	            IF ("gtyp_VGR".vertical_Axis.di_Actual_Position <= ("gtyp_VGR".di_Pos_Color_vertical + "gtyp_VGR".vertical_Axis.Config.di_Pos_Window))
	                AND ("gtyp_VGR".vertical_Axis.di_Actual_Position >= ("gtyp_VGR".di_Pos_Color_vertical - "gtyp_VGR".vertical_Axis.Config.di_Pos_Window))
	                AND "gtyp_VGR".vertical_Axis.x_Position_Reached THEN
	                "gtyp_VGR".vertical_Axis.x_Start_Positioning := FALSE;
	                "gtyp_VGR".vertical_Axis.i_PWM := 800;
	                #li_StepCase := 750;
	            END_IF;

	        750: // evaluate color workpiece
	            #ls_Color := '';

	            IF "IW_SSC_ColorSensor_A1" >= "gtyp_SSC".w_Threshold_Red_Blue THEN
	 //               IF "IW_SSC_ColorSensor" > 16000 AND "IW_SSC_ColorSensor" < 17500 THEN
	                #ls_Color := 'BLUE';
	            ELSIF "IW_SSC_ColorSensor_A1" <= "gtyp_SSC".w_Threshold_White_Red THEN
	//            ELSIF "IW_SSC_ColorSensor" > 5000 AND "IW_SSC_ColorSensor" < 11000 THEN
	                #ls_Color := 'WHITE';
	            ELSIF "IW_SSC_ColorSensor_A1" > "gtyp_SSC".w_Threshold_White_Red AND "IW_SSC_ColorSensor_A1" < "gtyp_SSC".w_Threshold_Red_Blue THEN
	//            ELSIF "IW_SSC_ColorSensor" > 11000 AND "IW_SSC_ColorSensor" < 16000 THEN
	                #ls_Color := 'RED';
	            END_IF;

	            #li_Return_LDT := RD_SYS_T(#ldt_MQTT);
	            "gtyp_VGR".History[2].ldt_ts := DT_TO_LDT(#ldt_MQTT);
	            "gtyp_VGR".History[2].i_code := 200;
	            "gtyp_VGR".Workpiece.s_type  := #ls_Color;

	            #lx_Start_TON_Wait  := TRUE;
	            #lt_TON_Wait        := T#500ms;

	            IF #lfb_TON_Wait.Q THEN
	                #lx_Start_TON_Wait := FALSE;
	                #li_StepCase := 760;
	            END_IF;

	        760: // Position vertical pre NFC
	            "gtyp_VGR".vertical_Axis.di_Target_Position := "gtyp_VGR".di_Pos_NFC_vertical - "gtyp_VGR".di_Offset_Pos_DSI_NFC_vertical;
	            "gtyp_VGR".vertical_Axis.x_Start_Positioning := TRUE;
	            "gtyp_VGR".vertical_Axis.i_PWM := 500;

	            IF ("gtyp_VGR".vertical_Axis.di_Actual_Position <= ("gtyp_VGR".di_Pos_NFC_vertical - "gtyp_VGR".di_Offset_Pos_DSI_NFC_vertical + "gtyp_VGR".vertical_Axis.Config.di_Pos_Window))
	                AND ("gtyp_VGR".vertical_Axis.di_Actual_Position >= ("gtyp_VGR".di_Pos_NFC_vertical - "gtyp_VGR".di_Offset_Pos_DSI_NFC_vertical - "gtyp_VGR".vertical_Axis.Config.di_Pos_Window))
	                AND "gtyp_VGR".vertical_Axis.x_Position_Reached THEN
	                "gtyp_VGR".vertical_Axis.x_Start_Positioning := FALSE;
	                "gtyp_VGR".vertical_Axis.i_PWM := 800;
	                #li_StepCase := 770;
	            END_IF;

	        770: // wait sequence
	            #lx_Start_TON_Wait := TRUE;
	            #lt_TON_Wait := T#500ms;

	            IF #lfb_TON_Wait.Q THEN
	                #lx_Start_TON_Wait := FALSE;
	                #li_StepCase := 780;
	            END_IF;

	        780: // Position horizontal/rotate NFC

	            "gtyp_VGR".horizontal_Axis.di_Target_Position := "gtyp_VGR".di_Pos_NFC_horizontal;
	            "gtyp_VGR".horizontal_Axis.x_Start_Positioning := TRUE;
	            "gtyp_VGR".rotate_Axis.di_Target_Position := "gtyp_VGR".di_Pos_NFC_rotate;
	            "gtyp_VGR".rotate_Axis.x_Start_Positioning := TRUE;

	            IF ("gtyp_VGR".horizontal_Axis.di_Actual_Position <= ("gtyp_VGR".di_Pos_NFC_horizontal + "gtyp_VGR".horizontal_Axis.Config.di_Pos_Window))
	                AND ("gtyp_VGR".horizontal_Axis.di_Actual_Position >= ("gtyp_VGR".di_Pos_NFC_horizontal - "gtyp_VGR".horizontal_Axis.Config.di_Pos_Window))
	                AND "gtyp_VGR".horizontal_Axis.x_Position_Reached THEN
	                "gtyp_VGR".horizontal_Axis.x_Start_Positioning := FALSE;
	            END_IF;

	            IF ("gtyp_VGR".rotate_Axis.di_Actual_Position <= ("gtyp_VGR".di_Pos_NFC_rotate + "gtyp_VGR".rotate_Axis.Config.di_Pos_Window))
	                AND ("gtyp_VGR".rotate_Axis.di_Actual_Position >= ("gtyp_VGR".di_Pos_NFC_rotate - "gtyp_VGR".rotate_Axis.Config.di_Pos_Window))
	                AND "gtyp_VGR".rotate_Axis.x_Position_Reached THEN
	                "gtyp_VGR".rotate_Axis.x_Start_Positioning := FALSE;
	            END_IF;

	            IF ("gtyp_VGR".horizontal_Axis.di_Actual_Position <= ("gtyp_VGR".di_Pos_NFC_horizontal + "gtyp_VGR".horizontal_Axis.Config.di_Pos_Window))
	                AND ("gtyp_VGR".horizontal_Axis.di_Actual_Position >= ("gtyp_VGR".di_Pos_NFC_horizontal - "gtyp_VGR".horizontal_Axis.Config.di_Pos_Window))
	                AND "gtyp_VGR".horizontal_Axis.x_Position_Reached
	                AND ("gtyp_VGR".rotate_Axis.di_Actual_Position <= ("gtyp_VGR".di_Pos_NFC_rotate + "gtyp_VGR".rotate_Axis.Config.di_Pos_Window))
	                AND ("gtyp_VGR".rotate_Axis.di_Actual_Position >= ("gtyp_VGR".di_Pos_NFC_rotate - "gtyp_VGR".rotate_Axis.Config.di_Pos_Window))
	                AND "gtyp_VGR".rotate_Axis.x_Position_Reached THEN
	                "gtyp_VGR".horizontal_Axis.x_Start_Positioning := FALSE;
	                "gtyp_VGR".vertical_Axis.x_Start_Positioning := FALSE;
	                "gtyp_VGR".rotate_Axis.x_Start_Positioning := FALSE;
	                #li_StepCase := 790;
	            END_IF;

	        790: // wait sequence
	            #lx_Start_TON_Wait := TRUE;
	            #lt_TON_Wait := T#500ms;

	            IF #lfb_TON_Wait.Q THEN
	                #lx_Start_TON_Wait := FALSE;
	                #li_StepCase := 800;
	            END_IF;

	        800: // Position vertical NFC

	            "gtyp_VGR".vertical_Axis.di_Target_Position := "gtyp_VGR".di_Pos_NFC_vertical;
	            "gtyp_VGR".vertical_Axis.x_Start_Positioning := TRUE;
	            "gtyp_VGR".vertical_Axis.i_PWM := 500;

	            IF ("gtyp_VGR".vertical_Axis.di_Actual_Position <= ("gtyp_VGR".di_Pos_NFC_vertical + "gtyp_VGR".vertical_Axis.Config.di_Pos_Window))
	                AND ("gtyp_VGR".vertical_Axis.di_Actual_Position >= ("gtyp_VGR".di_Pos_NFC_vertical - "gtyp_VGR".vertical_Axis.Config.di_Pos_Window))
	                AND "gtyp_VGR".vertical_Axis.x_Position_Reached THEN
	                "gtyp_VGR".vertical_Axis.x_Start_Positioning := FALSE;
	                "gtyp_VGR".vertical_Axis.i_PWM := 800;
	                #li_StepCase := 810;
	            END_IF;

	        810: // Start write/read NFC Color

	            "gtyp_VGR".x_NFC_Start := TRUE;

	            IF "gtyp_VGR".x_NFC_Completed THEN
	                "gtyp_VGR".x_NFC_Start := FALSE;
	                #li_StepCase := 820;
	            END_IF;

	        820: // Position vertical pre NFC

	            "gtyp_VGR".vertical_Axis.di_Target_Position := "gtyp_VGR".di_Pos_NFC_vertical - "gtyp_VGR".di_Offset_Pos_DSI_NFC_vertical;
	            "gtyp_VGR".vertical_Axis.x_Start_Positioning := TRUE;
	            "gtyp_VGR".vertical_Axis.i_PWM := 500;

	            IF ("gtyp_VGR".vertical_Axis.di_Actual_Position <= ("gtyp_VGR".di_Pos_NFC_vertical - "gtyp_VGR".di_Offset_Pos_DSI_NFC_vertical + "gtyp_VGR".vertical_Axis.Config.di_Pos_Window))
	                AND ("gtyp_VGR".vertical_Axis.di_Actual_Position >= ("gtyp_VGR".di_Pos_NFC_vertical - "gtyp_VGR".di_Offset_Pos_DSI_NFC_vertical - "gtyp_VGR".vertical_Axis.Config.di_Pos_Window))
	                AND "gtyp_VGR".vertical_Axis.x_Position_Reached THEN
	                "gtyp_VGR".vertical_Axis.x_Start_Positioning := FALSE;
	                "gtyp_VGR".vertical_Axis.i_PWM := 800;
	                #li_StepCase := 830;
	            END_IF;

	        830: // wait sequence
	            #lx_Start_TON_Wait := TRUE;
	            #lt_TON_Wait := T#500ms;

	            IF #lfb_TON_Wait.Q THEN
	                #lx_Start_TON_Wait := FALSE;
	                #li_StepCase := 840;
	            END_IF;

	        840: // Position rotate HBW and homing horizontal/vertical axis
	            "gtyp_VGR".rotate_Axis.di_Target_Position := "gtyp_VGR".di_Pos_HBW_rotate;
	            "gtyp_VGR".rotate_Axis.x_Start_Positioning := TRUE;

	            "gtyp_VGR".horizontal_Axis.x_Reference := TRUE;
	            "gtyp_VGR".vertical_Axis.x_Reference := TRUE;

	            IF ("gtyp_VGR".rotate_Axis.di_Actual_Position <= ("gtyp_VGR".di_Pos_HBW_rotate + "gtyp_VGR".rotate_Axis.Config.di_Pos_Window))
	                AND ("gtyp_VGR".rotate_Axis.di_Actual_Position >= ("gtyp_VGR".di_Pos_HBW_rotate - "gtyp_VGR".rotate_Axis.Config.di_Pos_Window))
	                AND "gtyp_VGR".rotate_Axis.x_Position_Reached THEN
	                "gtyp_VGR".rotate_Axis.x_Start_Positioning := FALSE;
	            END_IF;

	            IF NOT "gtyp_VGR".horizontal_Axis.x_Referenced AND NOT "gtyp_VGR".vertical_Axis.x_Referenced THEN
	                #li_StepCase := 850;
	            END_IF;

	        850: // Position rotate HBW reached and homed horizontal/vertical axis

	            IF ("gtyp_VGR".rotate_Axis.di_Actual_Position <= ("gtyp_VGR".di_Pos_HBW_rotate + "gtyp_VGR".rotate_Axis.Config.di_Pos_Window))
	                AND ("gtyp_VGR".rotate_Axis.di_Actual_Position >= ("gtyp_VGR".di_Pos_HBW_rotate - "gtyp_VGR".rotate_Axis.Config.di_Pos_Window))
	                AND "gtyp_VGR".rotate_Axis.x_Position_Reached THEN
	                "gtyp_VGR".rotate_Axis.x_Start_Positioning := FALSE;
	            END_IF;

	            IF "gtyp_VGR".horizontal_Axis.x_Referenced THEN
	                "gtyp_VGR".horizontal_Axis.x_Reference := FALSE;
	            END_IF;
	            IF "gtyp_VGR".vertical_Axis.x_Referenced THEN
	                "gtyp_VGR".vertical_Axis.x_Reference := FALSE;
	            END_IF;
	            IF "gtyp_VGR".horizontal_Axis.x_Referenced
	                AND "gtyp_VGR".vertical_Axis.x_Referenced
	                AND ("gtyp_VGR".rotate_Axis.di_Actual_Position <= ("gtyp_VGR".di_Pos_HBW_rotate + "gtyp_VGR".rotate_Axis.Config.di_Pos_Window))
	                AND ("gtyp_VGR".rotate_Axis.di_Actual_Position >= ("gtyp_VGR".di_Pos_HBW_rotate - "gtyp_VGR".rotate_Axis.Config.di_Pos_Window))
	                AND "gtyp_VGR".rotate_Axis.x_Position_Reached THEN
	                "gtyp_VGR".horizontal_Axis.x_Reference := FALSE;
	                "gtyp_VGR".vertical_Axis.x_Reference := FALSE;
	                "gtyp_VGR".rotate_Axis.x_Start_Positioning := FALSE;
	                #li_StepCase := 860;
	            END_IF;

	        860: // wait sequence
	            #lx_Start_TON_Wait := TRUE;
	            #lt_TON_Wait := T#500ms;

	            IF #lfb_TON_Wait.Q THEN
	                #lx_Start_TON_Wait := FALSE;
	                #li_StepCase := 870;
	            END_IF;

	        870: // Position horizontal HBW

	            "gtyp_VGR".horizontal_Axis.di_Target_Position := "gtyp_VGR".di_Pos_HBW_horizontal;
	            "gtyp_VGR".horizontal_Axis.x_Start_Positioning := TRUE;

	            IF ("gtyp_VGR".horizontal_Axis.di_Actual_Position <= ("gtyp_VGR".di_Pos_HBW_horizontal + "gtyp_VGR".horizontal_Axis.Config.di_Pos_Window))
	                AND ("gtyp_VGR".horizontal_Axis.di_Actual_Position >= ("gtyp_VGR".di_Pos_HBW_horizontal - "gtyp_VGR".horizontal_Axis.Config.di_Pos_Window))
	                AND "gtyp_VGR".horizontal_Axis.x_Position_Reached THEN
	                "gtyp_VGR".horizontal_Axis.x_Start_Positioning := FALSE;
	                #li_StepCase := 880;
	            END_IF;

	        880: // container available start drop down
	            IF "gtyp_HBW".x_HBW_Container_Available THEN
	                #li_StepCase := 890;
	            END_IF;

	        890: // Position vertical discard HBW
	            "gtyp_VGR".vertical_Axis.di_Target_Position := "gtyp_VGR".di_Pos_HBW_Discard_vertical;
	            "gtyp_VGR".vertical_Axis.x_Start_Positioning := TRUE;
	            "gtyp_VGR".vertical_Axis.i_PWM := 500;

	            IF ("gtyp_VGR".vertical_Axis.di_Actual_Position <= ("gtyp_VGR".di_Pos_HBW_Discard_vertical + "gtyp_VGR".vertical_Axis.Config.di_Pos_Window))
	                AND ("gtyp_VGR".vertical_Axis.di_Actual_Position >= ("gtyp_VGR".di_Pos_HBW_Discard_vertical - "gtyp_VGR".vertical_Axis.Config.di_Pos_Window))
	                AND "gtyp_VGR".vertical_Axis.x_Position_Reached THEN
	                "gtyp_VGR".vertical_Axis.x_Start_Positioning := FALSE;
	                "gtyp_VGR".vertical_Axis.i_PWM := 800;
	                #li_StepCase := 900;
	            END_IF;

	        900: // turn off vacuum
	            "QX_VGR_ValveVacuum_Q8" := FALSE;
	            #li_StepCase := 910;

	        910: // turn off compressor
	            "QX_VGR_Compressor_Q7" := FALSE;
	            "gtyp_VGR".x_HBW_Discards := TRUE;

	            #lx_Start_TON_Wait := TRUE;
	            #lt_TON_Wait := T#500ms;

	            IF #lfb_TON_Wait.Q AND "gtyp_HBW".x_HBW_Discards_Accepted THEN
	                #lx_State_activ := FALSE;
	                #ls_Target := '';
	                "gtyp_VGR".x_HBW_Discards   := FALSE;
	                "gtyp_VGR".x_HBW_Storage  := FALSE;
	                #lx_Start_TON_Wait                   := FALSE;
	                #li_StepCase                := 920;
	            END_IF;

	        920: // homing vertical axis
	            "gtyp_VGR".vertical_Axis.x_Reference := TRUE;

	            IF NOT "gtyp_VGR".vertical_Axis.x_Referenced THEN
	                #li_StepCase := 930;
	            END_IF;

	        930: // homed vertical axis
	            IF "gtyp_VGR".vertical_Axis.x_Referenced THEN
	                "gtyp_VGR".vertical_Axis.x_Reference := FALSE;
	                #li_StepCase := 940;
	            END_IF;

	        940: // homing horizontal axis
	            "gtyp_VGR".horizontal_Axis.x_Reference := TRUE;

	            IF NOT "gtyp_VGR".horizontal_Axis.x_Referenced THEN
	                #li_StepCase := 950;
	            END_IF;

	        950: // homed horizontal axis
	            IF "gtyp_VGR".horizontal_Axis.x_Referenced THEN
	                "gtyp_VGR".horizontal_Axis.x_Reference := FALSE;
	                #li_StepCase := 960;
	            END_IF;

	        960: // wait sequence
	            #lx_Start_TON_Wait := TRUE;
	            #lt_TON_Wait := T#500ms;

	            IF #lfb_TON_Wait.Q AND "gtyp_HBW".x_HBW_Discards_Accepted THEN
	                "gtyp_VGR".x_HBW_Discards  := FALSE;
	                #lx_Start_TON_Wait               := FALSE;
	                "gtyp_VGR".Workpiece.s_id       := '';
	                "gtyp_VGR".Workpiece.s_state    := '';
	                "gtyp_VGR".Workpiece.s_type     := '';
	                FOR #li_Counter := 1 TO 8 DO
	                    // Statement section FOR
	                    "gtyp_VGR".History[#li_Counter].i_code := 0;
	                    "gtyp_VGR".History[#li_Counter].ldt_ts := DT#1990-01-01-00:00:00;
	                END_FOR;
	                #li_StepCase := 0;
	            END_IF;

	        1200:// homing vertical axis
	            "gtyp_VGR".Workpiece.s_id := '0';
	            "gtyp_VGR".Workpiece.s_state := '';
	            "gtyp_VGR".Workpiece.s_type := '';
	            FOR #li_Counter := 1 TO 8 DO
	                "gtyp_VGR".History[#li_Counter].i_code := 0;
	                "gtyp_VGR".History[#li_Counter].ldt_ts := DT#1990-01-01-00:00:00;
	            END_FOR;

	            IF "gtyp_HBW".x_HBW_Container_Available THEN
	                "gtyp_VGR".x_HBW_Discards := TRUE;
	            END_IF;

	            IF "gtyp_HBW".x_HBW_Discards_Accepted OR "gtyp_HBW".x_HBW_PickedUp_Accepted THEN
	                "gtyp_VGR".x_HBW_Discards := FALSE;
	                "gtyp_VGR".x_HBW_PickedUp := FALSE;
	                "gtyp_HBW".x_HBW_Discards_Accepted := FALSE;
	                "gtyp_HBW".x_HBW_PickedUp_Accepted := FALSE;
	            END_IF;

	            #li_Lights := 2;
	            "gtyp_VGR".vertical_Axis.x_Reference := TRUE;

	            IF NOT "gtyp_VGR".vertical_Axis.x_Referenced THEN
	                #li_StepCase := 1210;
	            END_IF;

	        1210: // homed vertical axis
	            IF "gtyp_VGR".vertical_Axis.x_Referenced THEN
	                "gtyp_VGR".vertical_Axis.x_Reference := FALSE;
	                #li_StepCase := 1220;
	            END_IF;

	        1220: // homing horizontal axis
	            "gtyp_VGR".horizontal_Axis.x_Reference := TRUE;

	            IF NOT "gtyp_VGR".horizontal_Axis.x_Referenced THEN
	                #li_StepCase := 1230;
	            END_IF;

	        1230: // homed horizontal axis
	            IF "gtyp_VGR".horizontal_Axis.x_Referenced THEN
	                "gtyp_VGR".horizontal_Axis.x_Reference := FALSE;
	                #li_StepCase := 1240;
	            END_IF;

	        1240: // homing rotate axis
	            "gtyp_VGR".rotate_Axis.x_Reference := TRUE;

	            IF NOT "gtyp_VGR".rotate_Axis.x_Referenced THEN
	                #li_StepCase := 1250;
	            END_IF;

	        1250: // homed horizontal axis
	            IF "gtyp_VGR".rotate_Axis.x_Referenced THEN
	                "gtyp_VGR".rotate_Axis.x_Reference := FALSE;
	                #li_StepCase := 1260;
	            END_IF;

	        1260: // Position vertical/horizontal/rotate NiO
	            "gtyp_VGR".horizontal_Axis.di_Target_Position := "gtyp_VGR".di_Pos_NiO_horizontal;
	            "gtyp_VGR".horizontal_Axis.x_Start_Positioning := TRUE;
	            "gtyp_VGR".vertical_Axis.di_Target_Position := "gtyp_VGR".di_Pos_NiO_vertical;
	            "gtyp_VGR".vertical_Axis.x_Start_Positioning := TRUE;
	            "gtyp_VGR".vertical_Axis.i_PWM := 500;
	            "gtyp_VGR".rotate_Axis.di_Target_Position := "gtyp_VGR".di_Pos_NiO_rotate;
	            "gtyp_VGR".rotate_Axis.x_Start_Positioning := TRUE;

	            IF ("gtyp_VGR".horizontal_Axis.di_Actual_Position <= ("gtyp_VGR".di_Pos_NiO_horizontal + "gtyp_VGR".horizontal_Axis.Config.di_Pos_Window))
	                AND ("gtyp_VGR".horizontal_Axis.di_Actual_Position >= ("gtyp_VGR".di_Pos_NiO_horizontal - "gtyp_VGR".horizontal_Axis.Config.di_Pos_Window))
	                AND "gtyp_VGR".horizontal_Axis.x_Position_Reached THEN
	                "gtyp_VGR".horizontal_Axis.x_Start_Positioning := FALSE;
	            END_IF;

	            IF ("gtyp_VGR".vertical_Axis.di_Actual_Position <= ("gtyp_VGR".di_Pos_NiO_vertical + "gtyp_VGR".vertical_Axis.Config.di_Pos_Window))
	                AND ("gtyp_VGR".vertical_Axis.di_Actual_Position >= ("gtyp_VGR".di_Pos_NiO_vertical - "gtyp_VGR".vertical_Axis.Config.di_Pos_Window))
	                AND "gtyp_VGR".vertical_Axis.x_Position_Reached THEN
	                "gtyp_VGR".vertical_Axis.x_Start_Positioning := FALSE;
	            END_IF;

	            IF ("gtyp_VGR".rotate_Axis.di_Actual_Position <= ("gtyp_VGR".di_Pos_NiO_rotate + "gtyp_VGR".rotate_Axis.Config.di_Pos_Window))
	                AND ("gtyp_VGR".rotate_Axis.di_Actual_Position >= ("gtyp_VGR".di_Pos_NiO_rotate - "gtyp_VGR".rotate_Axis.Config.di_Pos_Window))
	                AND "gtyp_VGR".rotate_Axis.x_Position_Reached THEN
	                "gtyp_VGR".rotate_Axis.x_Start_Positioning := FALSE;
	            END_IF;

	            IF ("gtyp_VGR".horizontal_Axis.di_Actual_Position <= ("gtyp_VGR".di_Pos_NiO_horizontal + "gtyp_VGR".horizontal_Axis.Config.di_Pos_Window))
	                AND ("gtyp_VGR".horizontal_Axis.di_Actual_Position >= ("gtyp_VGR".di_Pos_NiO_horizontal - "gtyp_VGR".horizontal_Axis.Config.di_Pos_Window))
	                AND "gtyp_VGR".horizontal_Axis.x_Position_Reached
	                AND ("gtyp_VGR".vertical_Axis.di_Actual_Position <= ("gtyp_VGR".di_Pos_NiO_vertical + "gtyp_VGR".vertical_Axis.Config.di_Pos_Window))
	                AND ("gtyp_VGR".vertical_Axis.di_Actual_Position >= ("gtyp_VGR".di_Pos_NiO_vertical - "gtyp_VGR".vertical_Axis.Config.di_Pos_Window))
	                AND "gtyp_VGR".vertical_Axis.x_Position_Reached
	                AND ("gtyp_VGR".rotate_Axis.di_Actual_Position <= ("gtyp_VGR".di_Pos_NiO_rotate + "gtyp_VGR".rotate_Axis.Config.di_Pos_Window))
	                AND ("gtyp_VGR".rotate_Axis.di_Actual_Position >= ("gtyp_VGR".di_Pos_NiO_rotate - "gtyp_VGR".rotate_Axis.Config.di_Pos_Window))
	                AND "gtyp_VGR".rotate_Axis.x_Position_Reached THEN
	                "gtyp_VGR".horizontal_Axis.x_Start_Positioning := FALSE;
	                "gtyp_VGR".vertical_Axis.x_Start_Positioning := FALSE;
	                "gtyp_VGR".rotate_Axis.x_Start_Positioning := FALSE;
	                "gtyp_VGR".vertical_Axis.i_PWM := 800;
	                #li_StepCase := 1270;
	            END_IF;

	        1270: // turn off vacuum
	            "QX_VGR_ValveVacuum_Q8" := FALSE;
	            #li_StepCase := 1280;

	        1280: // turn off compressor

	            #lx_Start_TON_Wait := TRUE;
	            #lt_TON_Wait := T#1000ms;

	            IF #lfb_TON_Wait.Q THEN
	                "QX_VGR_Compressor_Q7"  := FALSE;
	                #lx_Start_TON_Wait               := FALSE;
	                "gtyp_VGR".x_Workpiece_NiO := FALSE;
	                "gtyp_VGR".x_HBW_Discards := FALSE;
	                #li_Lights := 1;
	                #li_StepCase            := 0;
	            END_IF;
	    // Statement section ELSE
	    ELSE
	            ;
	    END_CASE;

	ELSE
	    "gtyp_VGR".Workpiece.s_id := '';
	    "gtyp_VGR".Workpiece.s_state := '';
	    "gtyp_VGR".Workpiece.s_type := '';
	    // Order State
	    "gtyp_VGR".x_State_Process := FALSE;
	    "gtyp_Interface_Dashboard".Subscribe.State_Order.ldt_ts := DT_TO_LDT(#ldt_MQTT);
	    "gtyp_Interface_Dashboard".Subscribe.State_Order.s_state := 'WAITING_FOR_ORDER';
	    "gtyp_Interface_Dashboard".Subscribe.State_Order.s_type := '';
	    FOR #li_Counter := 1 TO 8 DO
	        "gtyp_VGR".History[#li_Counter].i_code := 0;
	        "gtyp_VGR".History[#li_Counter].ldt_ts := DT#1990-01-01-00:00:00;
	    END_FOR;

	    "gtyp_VGR".x_Start_Park_Position    := FALSE;
	    "gtyp_VGR".x_Park_Position_Reached  := FALSE;
	    "gtyp_VGR".x_NFC_Start_First        := FALSE;
	    "gtyp_VGR".x_NFC_Start              := FALSE;
	    "gtyp_VGR".x_NFC_Completed          := FALSE;
	    "gtyp_VGR".x_HBW_Storage            := FALSE;
	    "gtyp_VGR".x_HBW_Outsource          := FALSE;
	    "gtyp_VGR".s_HBW_Outsource_Typ      := '';
	    "gtyp_VGR".x_HBW_Discards           := FALSE;
	    "gtyp_VGR".x_HBW_PickedUp           := FALSE;
	    "gtyp_VGR".x_MPO_Req_Discard        := FALSE;
	    "gtyp_VGR".x_MPO_Discards           := FALSE;
	    "gtyp_VGR".x_Ready_For_Outsource    := FALSE;
	    "gtyp_VGR".x_State_Process          := FALSE;
	    "gtyp_VGR".x_Workpiece_NiO          := FALSE;

	    "gtyp_VGR".vertical_Axis.i_PWM      := 800;

	    #li_Lights := 1;
	    #lx_Init := TRUE;
	END_IF;
END_FUNCTION_BLOCK

FUNCTION_BLOCK "PRG_Order"
TITLE = Program Order
{ S7_Optimized_Access := 'TRUE' }
AUTHOR : 'A.Schaefer'
VERSION : 0.0
   VAR
      lx_Init { ExternalAccessible := 'False'; ExternalVisible := 'False'; ExternalWritable := 'False'} : Bool;
      li_StepCase { ExternalAccessible := 'False'; ExternalVisible := 'False'; ExternalWritable := 'False'} : Int;
      lldt_ts_old { ExternalAccessible := 'False'; ExternalVisible := 'False'; ExternalWritable := 'False'} : LDT;
      ldt_MQTT { ExternalAccessible := 'False'; ExternalVisible := 'False'; ExternalWritable := 'False'} : Date_And_Time;
      li_Return_LDT { ExternalAccessible := 'False'; ExternalVisible := 'False'; ExternalWritable := 'False'} : Int;
      lfb_TON_Wait {InstructionName := 'TON_TIME'; LibVersion := '1.0'; ExternalAccessible := 'False'; ExternalVisible := 'False'; ExternalWritable := 'False'; S7_SetPoint := 'False'} : TON_TIME;
      lx_Start_TON_Wait { ExternalAccessible := 'False'; ExternalVisible := 'False'; ExternalWritable := 'False'} : Bool;
   END_VAR


BEGIN
	IF #lx_Init THEN
	    #lfb_TON_Wait(IN:= #lx_Start_TON_Wait,PT:= T#20s);

	    // step chain order
	    CASE #li_StepCase OF

	        0:  // init
	            #lx_Start_TON_Wait := FALSE;
	            #li_StepCase := 10;

	        10: // check whether order button has been pressed (time stamp changes)
	            IF ("gtyp_Interface_Dashboard".Publish.OrderWorkpieceButton.ldt_ts > #lldt_ts_old) THEN
	                #li_Return_LDT := RD_SYS_T(#ldt_MQTT);
	                "gtyp_Interface_Dashboard".Subscribe.State_Order.ldt_ts := DT_TO_LDT(#ldt_MQTT);
	                "gtyp_Interface_Dashboard".Subscribe.State_Order.s_state := 'ORDERED';
	                "gtyp_VGR".s_HBW_Outsource_Typ := "gtyp_Interface_Dashboard".Publish.OrderWorkpieceButton.s_type;
	                "gtyp_Interface_Dashboard".Subscribe.State_Order.s_type := "gtyp_VGR".s_HBW_Outsource_Typ;
	                IF "gtyp_VGR".x_Ready_For_Outsource THEN
	                    #lldt_ts_old := "gtyp_Interface_Dashboard".Publish.OrderWorkpieceButton.ldt_ts;
	                    "gtyp_VGR".x_HBW_Outsource := TRUE;
	                    #li_StepCase := 20;
	                END_IF;
	            END_IF;

	        20: // delete
	            IF "gtyp_VGR".x_HBW_PickedUp OR NOT "gtyp_VGR".x_HBW_Outsource THEN
	                "gtyp_VGR".x_HBW_Outsource := FALSE;
	                "gtyp_VGR".s_HBW_Outsource_Typ := '';
	                #li_StepCase := 0;
	            END_IF;

	    // Statement section ELSE
	    ELSE
	                ;
	    END_CASE;

	ELSE
	    #lx_Init    := TRUE;
	    #lldt_ts_old:= LDT#1970-01-01-00:00:00;
	END_IF;
END_FUNCTION_BLOCK

FUNCTION_BLOCK "PRG_MPO_Set_Park_Position"
TITLE = Program Set Positioning HBW
{ S7_Optimized_Access := 'TRUE' }
AUTHOR : 'A.Schaefer'
VERSION : 0.0
   VAR
      lx_Init { ExternalAccessible := 'False'; ExternalVisible := 'False'; ExternalWritable := 'False'} : Bool;
      lx_Start_TON_Wait { ExternalAccessible := 'False'; ExternalVisible := 'False'; ExternalWritable := 'False'} : Bool;
      lt_TON_Wait { ExternalAccessible := 'False'; ExternalVisible := 'False'; ExternalWritable := 'False'} : Time;
      li_StepCase { ExternalAccessible := 'False'; ExternalVisible := 'False'; ExternalWritable := 'False'} : Int;
      lfb_TON_Wait {InstructionName := 'TON_TIME'; LibVersion := '1.0'; ExternalAccessible := 'False'; ExternalVisible := 'False'; ExternalWritable := 'False'; S7_SetPoint := 'False'} : TON_TIME;
      lfb_R_Trig_Start_Park_Pos {InstructionName := 'R_TRIG'; LibVersion := '1.0'; ExternalAccessible := 'False'; ExternalVisible := 'False'; ExternalWritable := 'False'; S7_SetPoint := 'False'} : R_TRIG;
   END_VAR


BEGIN
	IF #lx_Init THEN

	    // FB TON Wait
	    #lfb_TON_Wait(IN := #lx_Start_TON_Wait,
	                  PT := #lt_TON_Wait);

	    #lfb_R_Trig_Start_Park_Pos(CLK := "gtyp_Setup".x_Park_Position
	                               OR "IX_Set_Park_Position");

	    // Set Start Park Position
	    IF #lfb_R_Trig_Start_Park_Pos.Q THEN
	        "gtyp_MPO".x_Start_Park_Position := TRUE;
	        #li_StepCase := 0;
	    END_IF;

	    // not Start Park Pos Step 0
	    IF NOT "gtyp_MPO".x_Start_Park_Position THEN
	        #li_StepCase := 0;
	    END_IF;

	    // step chain HBW
	    CASE #li_StepCase OF

	        0:  // init
	            #lx_Start_TON_Wait := FALSE;
	            #li_StepCase := 10;

	        10:  // Set Positioning activ?
	            IF "gtyp_MPO".x_Start_Park_Position AND NOT "gtyp_MPO".x_Park_Position_Reached THEN
	                #li_StepCase := 20;
	            END_IF;

	        20: // Towards
	            "QX_MPO_M5_VacuumTowardsTurnTable_Q8" := FALSE;
	            "QX_MPO_M5_VacuumTowardsOven_Q7"    := TRUE;
	            #lx_Start_TON_Wait                  := TRUE;
	            #lt_TON_Wait                        := T#4000ms;

	            IF #lfb_TON_Wait.Q THEN
	                "QX_MPO_M5_VacuumTowardsTurnTable_Q8" := FALSE;
	                "QX_MPO_M5_VacuumTowardsOven_Q7"    := FALSE;
	                #lx_Start_TON_Wait                  := FALSE;
	                #li_StepCase                        := 30;
	            END_IF;

	        30: // homing vertical axis
	            "QX_MPO_M1_TurnTableClockwise_Q1"        := TRUE;
	            "QX_MPO_M1_TurnTableCounterclockwise_Q2" := FALSE;
	            #lx_Start_TON_Wait := TRUE;
	            #lt_TON_Wait := T#1000ms;

	            IF #lfb_TON_Wait.Q THEN
	                "QX_MPO_M1_TurnTableClockwise_Q1" := FALSE;
	                "QX_MPO_M1_TurnTableCounterclockwise_Q2" := FALSE;
	                #lx_Start_TON_Wait := FALSE;
	                #li_StepCase := 40;
	            END_IF;

	        40: // Deciding which doing
	            "gtyp_MPO".x_Park_Position_Reached := TRUE;


	            // Statement section ELSE
	        ELSE
	            ;
	    END_CASE;

	ELSE
	    #lx_Init := TRUE;
	END_IF;
END_FUNCTION_BLOCK

FUNCTION_BLOCK "PRG_HBW_Ablauf"
TITLE = Program Ablauf HBW
{ S7_Optimized_Access := 'TRUE' }
AUTHOR : 'A.Schaefer'
VERSION : 0.0
   VAR
      lx_Init { ExternalAccessible := 'False'; ExternalVisible := 'False'; ExternalWritable := 'False'} : Bool;
      lx_Start_TON_Wait { ExternalAccessible := 'False'; ExternalVisible := 'False'; ExternalWritable := 'False'} : Bool;
      lx_Time_Error { ExternalAccessible := 'False'; ExternalVisible := 'False'; ExternalWritable := 'False'} : Bool;
      lt_TON_Wait { ExternalAccessible := 'False'; ExternalVisible := 'False'; ExternalWritable := 'False'} : Time;
      lx_Start_TON_State { ExternalAccessible := 'False'; ExternalVisible := 'False'; ExternalWritable := 'False'} : Bool;
      lx_Storage { ExternalAccessible := 'False'; ExternalVisible := 'False'; ExternalWritable := 'False'} : Bool;
      ldt_MQTT { ExternalAccessible := 'False'; ExternalVisible := 'False'; ExternalWritable := 'False'} : Date_And_Time;
      li_Return_LDT { ExternalAccessible := 'False'; ExternalVisible := 'False'; ExternalWritable := 'False'} : Int;
      lldt_Outsource { ExternalAccessible := 'False'; ExternalVisible := 'False'; ExternalWritable := 'False'} : LDT;
      li_Lights { ExternalAccessible := 'False'; ExternalVisible := 'False'; ExternalWritable := 'False'} : Int;
      li_Lights_old { ExternalAccessible := 'False'; ExternalVisible := 'False'; ExternalWritable := 'False'} : Int;
      li_Counter_Hor { ExternalAccessible := 'False'; ExternalVisible := 'False'; ExternalWritable := 'False'} : Int;
      li_Counter_Ver { ExternalAccessible := 'False'; ExternalVisible := 'False'; ExternalWritable := 'False'} : Int;
      li_Counter_Act_Hor { ExternalAccessible := 'False'; ExternalVisible := 'False'; ExternalWritable := 'False'} : Int;
      li_Counter_Act_Ver { ExternalAccessible := 'False'; ExternalVisible := 'False'; ExternalWritable := 'False'} : Int;
      li_Counter { ExternalAccessible := 'False'; ExternalVisible := 'False'; ExternalWritable := 'False'} : Int;
      li_StepCase { ExternalAccessible := 'False'; ExternalVisible := 'False'; ExternalWritable := 'False'} : Int;
      ldi_PosRack_Horizontal { ExternalAccessible := 'False'; ExternalVisible := 'False'; ExternalWritable := 'False'} : DInt;
      ldi_PosRack_Vertical { ExternalAccessible := 'False'; ExternalVisible := 'False'; ExternalWritable := 'False'} : DInt;
      ls_Color { ExternalAccessible := 'False'; ExternalVisible := 'False'; ExternalWritable := 'False'} : String;
      lfb_TON_State {InstructionName := 'TON_TIME'; LibVersion := '1.0'; ExternalAccessible := 'False'; ExternalVisible := 'False'; ExternalWritable := 'False'; S7_SetPoint := 'False'} : TON_TIME;
      lfb_TON_ConveyerBelt_Out {InstructionName := 'TON_TIME'; LibVersion := '1.0'; ExternalAccessible := 'False'; ExternalVisible := 'False'; ExternalWritable := 'False'; S7_SetPoint := 'False'} : TON_TIME;
      lfb_TON_Wait {InstructionName := 'TON_TIME'; LibVersion := '1.0'; ExternalAccessible := 'False'; ExternalVisible := 'False'; ExternalWritable := 'False'; S7_SetPoint := 'False'} : TON_TIME;
      lfb_TON_Error {InstructionName := 'TON_TIME'; LibVersion := '1.0'; ExternalAccessible := 'False'; ExternalVisible := 'False'; ExternalWritable := 'False'; S7_SetPoint := 'False'} : TON_TIME;
   END_VAR


BEGIN
	IF #lx_Init THEN

	    // Restart after set Positioning
	    IF "gtyp_Setup".x_Set_Pos_Activ OR "gtyp_HBW".x_Start_Park_Position THEN
	        #li_StepCase := 0;
	    END_IF;

	    // wait time state
	    #lfb_TON_State(IN := NOT #lx_Start_TON_State,
	                    PT := T#2s);

	    // runtime monitoring error
	    #lfb_TON_Error(IN := #lx_Time_Error,
	                   PT := T#30s);

	    // state of the Stock HBW cyclically transmitted to the cloud
	     IF (#lfb_TON_State.Q OR (#li_Lights <> #li_Lights_old)) AND NOT #lx_Start_TON_State THEN
	        #li_Lights_old := #li_Lights;
	        #lx_Start_TON_State := TRUE;
	        #li_Return_LDT := RD_SYS_T(#ldt_MQTT);
	        "gtyp_Interface_Dashboard".Subscribe.Stock_HBW.StockItem := "gtyp_HBW".Rack_Workpiece;
	        "gtyp_Interface_Dashboard".Subscribe.Stock_HBW.ldt_ts := DT_TO_LDT(#ldt_MQTT);

	        "gtyp_Interface_Dashboard".Subscribe.State_HBW.ldt_ts := DT_TO_LDT(#ldt_MQTT);
	        "gtyp_Interface_Dashboard".Subscribe.State_HBW.i_code := #li_Lights;
	        "gtyp_Interface_Dashboard".Subscribe.State_HBW.s_description := '';
	        "gtyp_Interface_Dashboard".Subscribe.State_HBW.s_station := 'hbw';
	        "gtyp_Interface_Dashboard".Subscribe.State_HBW.s_target := '';
	    END_IF;

	    // restart wait time state
	    IF NOT #lfb_TON_State.Q AND #lx_Start_TON_State THEN
	        #lx_Start_TON_State := FALSE;
	    END_IF;

	    // FB TON Wait
	    #lfb_TON_Wait(IN := #lx_Start_TON_Wait,
	                    PT := #lt_TON_Wait);

	    //Run-on time Conveyer Belt
	    #lfb_TON_ConveyerBelt_Out(IN := NOT "IX_HBW_LightBarrierOutside_I3",
	                              PT := T#300ms);

	    // Reload the calibration values - Rack Array
	    // A
	    "gtyp_HBW".Rack_Pos[1, 1].di_PosRack_Horizontal := "gtyp_HBW".di_PosRack_A1_Horizontal;
	    "gtyp_HBW".Rack_Pos[2, 1].di_PosRack_Horizontal := "gtyp_HBW".di_PosRack_A1_Horizontal;
	    "gtyp_HBW".Rack_Pos[3, 1].di_PosRack_Horizontal := "gtyp_HBW".di_PosRack_A1_Horizontal;
	    // B
	    "gtyp_HBW".Rack_Pos[1, 2].di_PosRack_Horizontal := "gtyp_HBW".di_PosRack_B2_Horizontal;
	    "gtyp_HBW".Rack_Pos[2, 2].di_PosRack_Horizontal := "gtyp_HBW".di_PosRack_B2_Horizontal;
	    "gtyp_HBW".Rack_Pos[3, 2].di_PosRack_Horizontal := "gtyp_HBW".di_PosRack_B2_Horizontal;
	    // C
	    "gtyp_HBW".Rack_Pos[1, 3].di_PosRack_Horizontal := "gtyp_HBW".di_PosRack_C3_Horizontal;
	    "gtyp_HBW".Rack_Pos[2, 3].di_PosRack_Horizontal := "gtyp_HBW".di_PosRack_C3_Horizontal;
	    "gtyp_HBW".Rack_Pos[3, 3].di_PosRack_Horizontal := "gtyp_HBW".di_PosRack_C3_Horizontal;
	    // 1
	    "gtyp_HBW".Rack_Pos[1, 1].di_PosRack_Vertical := "gtyp_HBW".di_PosRack_A1_Vertical;
	    "gtyp_HBW".Rack_Pos[1, 2].di_PosRack_Vertical := "gtyp_HBW".di_PosRack_A1_Vertical;
	    "gtyp_HBW".Rack_Pos[1, 3].di_PosRack_Vertical := "gtyp_HBW".di_PosRack_A1_Vertical;
	    // 2
	    "gtyp_HBW".Rack_Pos[2, 1].di_PosRack_Vertical := "gtyp_HBW".di_PosRack_B2_Vertical;
	    "gtyp_HBW".Rack_Pos[2, 2].di_PosRack_Vertical := "gtyp_HBW".di_PosRack_B2_Vertical;
	    "gtyp_HBW".Rack_Pos[2, 3].di_PosRack_Vertical := "gtyp_HBW".di_PosRack_B2_Vertical;
	    // 3
	    "gtyp_HBW".Rack_Pos[3, 1].di_PosRack_Vertical := "gtyp_HBW".di_PosRack_C3_Vertical;
	    "gtyp_HBW".Rack_Pos[3, 2].di_PosRack_Vertical := "gtyp_HBW".di_PosRack_C3_Vertical;
	    "gtyp_HBW".Rack_Pos[3, 3].di_PosRack_Vertical := "gtyp_HBW".di_PosRack_C3_Vertical;

	    // step chain HBW
	    CASE #li_StepCase OF

	        0:  // init
	            #lx_Start_TON_Wait := FALSE;
	            #lx_Time_Error := FALSE;

	            "gtyp_HBW".Horizontal_Axis.x_Start_Positioning := FALSE;
	            "gtyp_HBW".Vertical_Axis.x_Start_Positioning := FALSE;
	            "gtyp_HBW".Horizontal_Axis.x_Reference := FALSE;
	            "gtyp_HBW".Vertical_Axis.x_Reference := FALSE;

	            IF NOT "gtyp_HBW".x_Error AND NOT "gtyp_Setup".x_Set_Pos_Activ AND NOT "gtyp_HBW".x_Start_Park_Position THEN
	                #li_StepCase := 10;
	            END_IF;

	        10:  // Position Cantilever Back
	            #li_Lights := 2;
	            IF "IX_HBW_SwitchCantileverFront_I5" OR NOT "IX_HBW_SwitchCantileverBack_I6" THEN
	                "QX_HBW_M4_CantileverBackward_Q8" := TRUE;
	                "QX_HBW_M4_CantileverForward_Q7" := FALSE;
	            ELSIF NOT "IX_HBW_SwitchCantileverFront_I5" AND "IX_HBW_SwitchCantileverBack_I6" THEN
	                "QX_HBW_M4_CantileverBackward_Q8" := FALSE;
	                "QX_HBW_M4_CantileverForward_Q7" := FALSE;
	                #li_StepCase := 20;
	            END_IF;

	        20: //homing vertical/horizontal axis

	            "gtyp_HBW".Horizontal_Axis.x_Reference := TRUE;
	            "gtyp_HBW".Vertical_Axis.x_Reference := TRUE;

	            IF NOT "gtyp_HBW".Horizontal_Axis.x_Referenced AND NOT "gtyp_HBW".Vertical_Axis.x_Referenced THEN
	                #li_StepCase := 30;
	            END_IF;

	        30: // homed vertical/horizontal axis
	            IF "gtyp_HBW".Horizontal_Axis.x_Referenced THEN
	                "gtyp_HBW".Horizontal_Axis.x_Reference := FALSE;
	            END_IF;
	            IF "gtyp_HBW".Vertical_Axis.x_Referenced THEN
	                "gtyp_HBW".Vertical_Axis.x_Reference := FALSE;
	            END_IF;

	            IF "gtyp_HBW".Horizontal_Axis.x_Referenced AND "gtyp_HBW".Vertical_Axis.x_Referenced THEN
	                "gtyp_HBW".Horizontal_Axis.x_Reference := FALSE;
	                "gtyp_HBW".Vertical_Axis.x_Reference := FALSE;
	                #li_StepCase := 40;
	            END_IF;

	        40: // Deciding which route to take

	            #li_Lights := 1;
	            #lx_Storage := FALSE;

	            // Procedure - storage
	            IF "gtyp_VGR".x_HBW_Storage THEN
	                #li_Lights := 2;
	                #li_StepCase := 50;
	            // Procedure - outsource
	            ELSIF "gtyp_VGR".x_HBW_Outsource THEN
	                #li_Lights := 2;
	                #li_StepCase := 60;
	            END_IF;

	        50: // Evaluate the next free position in the high-bay warehouse
	            FOR #li_Counter_Hor := 1 TO 3 DO
	                FOR #li_Counter_Ver := 1 TO 3 DO
	                    IF "gtyp_HBW".Rack_Workpiece[#li_Counter_Ver, #li_Counter_Hor].s_id = '0' THEN
	                        #li_Counter_Act_Hor := #li_Counter_Hor;
	                        #li_Counter_Act_Ver := #li_Counter_Ver;
	                        #ldi_PosRack_Horizontal := "gtyp_HBW".Rack_Pos[#li_Counter_Ver, #li_Counter_Hor].di_PosRack_Horizontal;
	                        #ldi_PosRack_Vertical := "gtyp_HBW".Rack_Pos[#li_Counter_Ver, #li_Counter_Hor].di_PosRack_Vertical;
	                        #li_StepCase := 70;
	                    END_IF;
	                    IF #li_StepCase = 70 THEN
	                        EXIT;
	                    END_IF;
	                END_FOR;
	                IF #li_StepCase = 70 THEN
	                    EXIT;
	                END_IF;
	            END_FOR;

	        60: // Evaluate the workpiece first stored in the high-bay warehouse with the appropriate color
	            #li_Return_LDT := RD_SYS_T(#ldt_MQTT);
	            #lldt_Outsource := #ldt_MQTT;

	            FOR #li_Counter_Hor := 1 TO 3 DO
	                FOR #li_Counter_Ver := 1 TO 3 DO
	                    IF ("gtyp_VGR".s_HBW_Outsource_Typ = "gtyp_HBW".Rack_Workpiece[#li_Counter_Ver, #li_Counter_Hor].s_type)
	                        AND (#lldt_Outsource > "gtyp_HBW".Rack_History[#li_Counter_Ver, #li_Counter_Hor].History[3].ldt_ts)
	                        AND NOT ("gtyp_HBW".Rack_History[#li_Counter_Ver, #li_Counter_Hor].History[3].ldt_ts = LDT#1970-01-01-00:00:00) THEN
	                        #lldt_Outsource := "gtyp_HBW".Rack_History[#li_Counter_Ver, #li_Counter_Hor].History[3].ldt_ts;
	                        #li_Counter_Act_Hor := #li_Counter_Hor;
	                        #li_Counter_Act_Ver := #li_Counter_Ver;
	                        #ldi_PosRack_Horizontal := "gtyp_HBW".Rack_Pos[#li_Counter_Ver, #li_Counter_Hor].di_PosRack_Horizontal;
	                        #ldi_PosRack_Vertical := "gtyp_HBW".Rack_Pos[#li_Counter_Ver, #li_Counter_Hor].di_PosRack_Vertical;
	                    END_IF;
	                END_FOR;
	            END_FOR;

	            IF (#li_Counter_Act_Hor = 4) OR (#li_Counter_Act_Ver = 4) THEN
	                #li_StepCase := 40;
	            ELSE
	                #li_StepCase := 70;
	            END_IF;

	        70: // Position vertical/horizontal HBW
	            "gtyp_HBW".Horizontal_Axis.di_Target_Position := #ldi_PosRack_Horizontal;
	            "gtyp_HBW".Horizontal_Axis.x_Start_Positioning := TRUE;
	            "gtyp_HBW".Vertical_Axis.di_Target_Position := #ldi_PosRack_Vertical;
	            "gtyp_HBW".Vertical_Axis.x_Start_Positioning := TRUE;

	            IF ("gtyp_HBW".Horizontal_Axis.di_Actual_Position <= (#ldi_PosRack_Horizontal + "gtyp_HBW".Horizontal_Axis.Config.di_Pos_Window))
	                AND ("gtyp_HBW".Horizontal_Axis.di_Actual_Position >= (#ldi_PosRack_Horizontal - "gtyp_HBW".Horizontal_Axis.Config.di_Pos_Window))
	                AND "gtyp_HBW".Horizontal_Axis.x_Position_Reached THEN
	                "gtyp_HBW".Horizontal_Axis.x_Start_Positioning := FALSE;
	            END_IF;

	            IF ("gtyp_HBW".Vertical_Axis.di_Actual_Position <= (#ldi_PosRack_Vertical + "gtyp_HBW".Vertical_Axis.Config.di_Pos_Window))
	                AND ("gtyp_HBW".Vertical_Axis.di_Actual_Position >= (#ldi_PosRack_Vertical - "gtyp_HBW".Vertical_Axis.Config.di_Pos_Window))
	                AND "gtyp_HBW".Vertical_Axis.x_Position_Reached THEN
	                "gtyp_HBW".Vertical_Axis.x_Start_Positioning := FALSE;
	            END_IF;

	            IF ("gtyp_HBW".Horizontal_Axis.di_Actual_Position <= (#ldi_PosRack_Horizontal + "gtyp_HBW".Horizontal_Axis.Config.di_Pos_Window))
	                AND ("gtyp_HBW".Horizontal_Axis.di_Actual_Position >= (#ldi_PosRack_Horizontal - "gtyp_HBW".Horizontal_Axis.Config.di_Pos_Window))
	                AND "gtyp_HBW".Horizontal_Axis.x_Position_Reached
	                AND ("gtyp_HBW".Vertical_Axis.di_Actual_Position <= (#ldi_PosRack_Vertical + "gtyp_HBW".Vertical_Axis.Config.di_Pos_Window))
	                AND ("gtyp_HBW".Vertical_Axis.di_Actual_Position >= (#ldi_PosRack_Vertical - "gtyp_HBW".Vertical_Axis.Config.di_Pos_Window))
	                AND "gtyp_HBW".Vertical_Axis.x_Position_Reached THEN
	                "gtyp_HBW".Horizontal_Axis.x_Start_Positioning := FALSE;
	                "gtyp_HBW".Vertical_Axis.x_Start_Positioning := FALSE;
	                #li_StepCase := 80;
	            END_IF;

	        80: // Position Cantilever Forward HBW

	            "QX_HBW_M4_CantileverBackward_Q8" := FALSE;
	            "QX_HBW_M4_CantileverForward_Q7" := TRUE;

	            IF "IX_HBW_SwitchCantileverFront_I5" AND NOT "IX_HBW_SwitchCantileverBack_I6" THEN
	                "QX_HBW_M4_CantileverBackward_Q8" := FALSE;
	                "QX_HBW_M4_CantileverForward_Q7" := FALSE;
	                #li_StepCase := 90;
	            END_IF;

	        90: // Position vertical+offset HBW
	            "gtyp_HBW".Vertical_Axis.di_Target_Position := #ldi_PosRack_Vertical - "gtyp_HBW".di_Offset_Pos_Rack_Vertical;
	            "gtyp_HBW".Vertical_Axis.x_Start_Positioning := TRUE;

	            IF ("gtyp_HBW".Vertical_Axis.di_Actual_Position <= (#ldi_PosRack_Vertical - "gtyp_HBW".di_Offset_Pos_Rack_Vertical + "gtyp_HBW".Vertical_Axis.Config.di_Pos_Window))
	                AND ("gtyp_HBW".Vertical_Axis.di_Actual_Position >= (#ldi_PosRack_Vertical - "gtyp_HBW".di_Offset_Pos_Rack_Vertical - "gtyp_HBW".Vertical_Axis.Config.di_Pos_Window))
	                AND "gtyp_HBW".Vertical_Axis.x_Position_Reached THEN
	                "gtyp_HBW".Vertical_Axis.x_Start_Positioning := FALSE;
	                #li_StepCase := 100;
	            END_IF;

	        100: // Position vertical Back HBW

	            "QX_HBW_M4_CantileverBackward_Q8" := TRUE;
	            "QX_HBW_M4_CantileverForward_Q7" := FALSE;

	            IF NOT "IX_HBW_SwitchCantileverFront_I5" AND "IX_HBW_SwitchCantileverBack_I6" THEN
	                IF "gtyp_VGR".x_HBW_Storage THEN
	                    "gtyp_HBW".Rack_Workpiece[#li_Counter_Act_Ver, #li_Counter_Act_Hor].s_id := '';
	                ELSIF "gtyp_VGR".x_HBW_Outsource THEN
	                    "gtyp_Interface_Dashboard".Subscribe.State_HBW.x_active := TRUE;
	                    "gtyp_HBW".History := "gtyp_HBW".Rack_History[#li_Counter_Act_Ver, #li_Counter_Act_Hor].History;
	                    "gtyp_HBW".Workpiece := "gtyp_HBW".Rack_Workpiece[#li_Counter_Act_Ver, #li_Counter_Act_Hor];
	                    #li_Return_LDT := RD_SYS_T(#ldt_MQTT);
	                    "gtyp_HBW".History[4].i_code := 400;
	                    "gtyp_HBW".History[4].ldt_ts := DT_TO_LDT(#ldt_MQTT);

	                    "gtyp_HBW".Rack_Workpiece[#li_Counter_Act_Ver, #li_Counter_Act_Hor].s_id := '';
	                    "gtyp_HBW".Rack_Workpiece[#li_Counter_Act_Ver, #li_Counter_Act_Hor].s_state := '';
	                    "gtyp_HBW".Rack_Workpiece[#li_Counter_Act_Ver, #li_Counter_Act_Hor].s_type := '';
	                    FOR #li_Counter := 1 TO 8 DO
	                        "gtyp_HBW".Rack_History[#li_Counter_Act_Ver, #li_Counter_Act_Hor].History[#li_Counter].i_code := 0;
	                        "gtyp_HBW".Rack_History[#li_Counter_Act_Ver, #li_Counter_Act_Hor].History[#li_Counter].ldt_ts := DT#1990-01-01-00:00:00;
	                    END_FOR;
	                END_IF;
	                "QX_HBW_M4_CantileverBackward_Q8" := FALSE;
	                "QX_HBW_M4_CantileverForward_Q7" := FALSE;
	                #li_StepCase := 110;
	            END_IF;

	        110: // homing vertical/horizontal axis

	            "gtyp_HBW".Horizontal_Axis.x_Reference := TRUE;

	            "gtyp_HBW".Vertical_Axis.di_Target_Position := "gtyp_HBW".di_PosBelt_Vertical - "gtyp_HBW".di_Offset_Pos_Belt_Vertical;
	            "gtyp_HBW".Vertical_Axis.x_Start_Positioning := TRUE;

	            IF ("gtyp_HBW".Vertical_Axis.di_Actual_Position <= ("gtyp_HBW".di_PosBelt_Vertical - "gtyp_HBW".di_Offset_Pos_Belt_Vertical + "gtyp_HBW".Vertical_Axis.Config.di_Pos_Window))
	                AND ("gtyp_HBW".Vertical_Axis.di_Actual_Position >= ("gtyp_HBW".di_PosBelt_Vertical - "gtyp_HBW".di_Offset_Pos_Belt_Vertical - "gtyp_HBW".Vertical_Axis.Config.di_Pos_Window))
	                AND "gtyp_HBW".Vertical_Axis.x_Position_Reached THEN
	                "gtyp_HBW".Vertical_Axis.x_Start_Positioning := FALSE;
	            END_IF;

	            IF NOT "gtyp_HBW".Horizontal_Axis.x_Referenced THEN
	                #li_StepCase := 120;
	            END_IF;

	        120: //homed vertical/horizontal axis

	            IF "gtyp_HBW".Horizontal_Axis.x_Referenced THEN
	                "gtyp_HBW".Horizontal_Axis.x_Reference := FALSE;
	            END_IF;

	            IF ("gtyp_HBW".Vertical_Axis.di_Actual_Position <= ("gtyp_HBW".di_PosBelt_Vertical - "gtyp_HBW".di_Offset_Pos_Belt_Vertical + "gtyp_HBW".Vertical_Axis.Config.di_Pos_Window))
	                AND ("gtyp_HBW".Vertical_Axis.di_Actual_Position >= ("gtyp_HBW".di_PosBelt_Vertical - "gtyp_HBW".di_Offset_Pos_Belt_Vertical - "gtyp_HBW".Vertical_Axis.Config.di_Pos_Window))
	                AND "gtyp_HBW".Vertical_Axis.x_Position_Reached THEN
	                "gtyp_HBW".Vertical_Axis.x_Start_Positioning := FALSE;
	            END_IF;

	            IF "gtyp_HBW".Horizontal_Axis.x_Referenced
	                AND ("gtyp_HBW".Vertical_Axis.di_Actual_Position <= ("gtyp_HBW".di_PosBelt_Vertical - "gtyp_HBW".di_Offset_Pos_Belt_Vertical + "gtyp_HBW".Vertical_Axis.Config.di_Pos_Window))
	                AND ("gtyp_HBW".Vertical_Axis.di_Actual_Position >= ("gtyp_HBW".di_PosBelt_Vertical - "gtyp_HBW".di_Offset_Pos_Belt_Vertical - "gtyp_HBW".Vertical_Axis.Config.di_Pos_Window))
	                AND "gtyp_HBW".Vertical_Axis.x_Position_Reached  THEN
	                "gtyp_HBW".Horizontal_Axis.x_Reference := FALSE;
	                "gtyp_HBW".Vertical_Axis.x_Start_Positioning := FALSE;
	                #li_StepCase := 130;
	            END_IF;

	        130: // Position vertical+offset/horizontal Belt
	            "gtyp_HBW".Horizontal_Axis.di_Target_Position := "gtyp_HBW".di_PosBelt_Horizontal;
	            "gtyp_HBW".Horizontal_Axis.x_Start_Positioning := TRUE;

	            IF ("gtyp_HBW".Horizontal_Axis.di_Actual_Position <= ("gtyp_HBW".di_PosBelt_Horizontal + "gtyp_HBW".Horizontal_Axis.Config.di_Pos_Window))
	                AND ("gtyp_HBW".Horizontal_Axis.di_Actual_Position >= ("gtyp_HBW".di_PosBelt_Horizontal - "gtyp_HBW".Horizontal_Axis.Config.di_Pos_Window))
	                AND "gtyp_HBW".Horizontal_Axis.x_Position_Reached THEN
	                "gtyp_HBW".Horizontal_Axis.x_Start_Positioning := FALSE;
	            END_IF;

	            IF ("gtyp_HBW".Horizontal_Axis.di_Actual_Position <= ("gtyp_HBW".di_PosBelt_Horizontal + "gtyp_HBW".Horizontal_Axis.Config.di_Pos_Window))
	                AND ("gtyp_HBW".Horizontal_Axis.di_Actual_Position >= ("gtyp_HBW".di_PosBelt_Horizontal - "gtyp_HBW".Horizontal_Axis.Config.di_Pos_Window))
	                AND "gtyp_HBW".Horizontal_Axis.x_Position_Reached THEN
	                "gtyp_HBW".Horizontal_Axis.x_Start_Positioning := FALSE;
	                #li_StepCase := 140;
	            END_IF;

	        140: // Position cantilever Forward Belt

	            "QX_HBW_M4_CantileverBackward_Q8" := FALSE;
	            "QX_HBW_M4_CantileverForward_Q7" := TRUE;

	            #lx_Time_Error := TRUE;

	            IF "IX_HBW_SwitchCantileverFront_I5" AND NOT "IX_HBW_SwitchCantileverBack_I6" THEN
	                "QX_HBW_M4_CantileverBackward_Q8"   := FALSE;
	                "QX_HBW_M4_CantileverForward_Q7"    := FALSE;
	                #lx_Time_Error                      := FALSE;
	                #li_StepCase := 150;
	            END_IF;

	            // runtime error
	            IF #lfb_TON_Error.Q THEN
	                #li_Lights := 4;
	                #lx_Time_Error := FALSE;
	                "QX_HBW_M1_ConveyorBeltBackward_Q2" := FALSE;
	                "QX_HBW_M1_ConveyorBeltForward_Q1" := FALSE;
	                "gtyp_Interface_Dashboard".Subscribe.State_HBW.x_active := FALSE;
	                "gtyp_HBW".x_Error := TRUE;
	                #li_StepCase := 0;
	            END_IF;

	        150: // Position vertical Belt
	            "gtyp_HBW".Vertical_Axis.di_Target_Position := "gtyp_HBW".di_PosBelt_Vertical;
	            "gtyp_HBW".Vertical_Axis.x_Start_Positioning := TRUE;

	            IF ("gtyp_HBW".Vertical_Axis.di_Actual_Position <= ("gtyp_HBW".di_PosBelt_Vertical + "gtyp_HBW".Vertical_Axis.Config.di_Pos_Window))
	                AND ("gtyp_HBW".Vertical_Axis.di_Actual_Position >= ("gtyp_HBW".di_PosBelt_Vertical - "gtyp_HBW".Vertical_Axis.Config.di_Pos_Window))
	                AND "gtyp_HBW".Vertical_Axis.x_Position_Reached THEN
	                "gtyp_HBW".Vertical_Axis.x_Start_Positioning := FALSE;
	                #li_StepCase := 160;
	            END_IF;

	        160: // Start Conveyor Belt Forward

	            #lx_Time_Error := TRUE;

	            IF NOT "IX_HBW_LightBarrierInside_I2" THEN
	                "QX_HBW_M1_ConveyorBeltBackward_Q2" := FALSE;
	                "QX_HBW_M1_ConveyorBeltForward_Q1"  := TRUE;
	                #lx_Time_Error                      := FALSE;
	                #li_StepCase                        := 170;
	            END_IF;

	            // runtime error
	            IF #lfb_TON_Error.Q THEN
	                #li_Lights := 4;
	                #lx_Time_Error := FALSE;
	                "QX_HBW_M1_ConveyorBeltBackward_Q2" := FALSE;
	                "QX_HBW_M1_ConveyorBeltForward_Q1" := FALSE;
	                "gtyp_Interface_Dashboard".Subscribe.State_HBW.x_active := FALSE;
	                "gtyp_HBW".x_Error := TRUE;
	                #li_StepCase := 0;
	            END_IF;

	        170: //Run-on time reached Conveyor Belt Outside

	            #lx_Time_Error := TRUE;

	            IF #lfb_TON_ConveyerBelt_Out.Q THEN
	                "QX_HBW_M1_ConveyorBeltBackward_Q2" := FALSE;
	                "QX_HBW_M1_ConveyorBeltForward_Q1" := FALSE;
	                "gtyp_HBW".x_HBW_Container_Available := TRUE;
	                #lx_Time_Error := FALSE;
	                #li_StepCase := 180;
	            END_IF;

	            // runtime error
	            IF #lfb_TON_Error.Q THEN
	                #li_Lights := 4;
	                #lx_Time_Error := FALSE;
	                "QX_HBW_M1_ConveyorBeltBackward_Q2" := FALSE;
	                "QX_HBW_M1_ConveyorBeltForward_Q1" := FALSE;
	                "gtyp_Interface_Dashboard".Subscribe.State_HBW.x_active := FALSE;
	                "gtyp_HBW".x_Error := TRUE;
	                #li_StepCase := 0;
	            END_IF;

	        180: // VGR picked up - outsource

	            #li_Lights := 1;

	            IF "gtyp_VGR".x_HBW_PickedUp AND "gtyp_VGR".x_HBW_Outsource THEN
	                "gtyp_VGR".Workpiece := "gtyp_HBW".Workpiece;
	                "gtyp_VGR".History   := "gtyp_HBW".History;
	                "gtyp_HBW".Workpiece.s_id := '0';
	                "gtyp_HBW".Workpiece.s_state := '';
	                "gtyp_HBW".Workpiece.s_type := '';
	                FOR #li_Counter := 1 TO 8 DO
	                    "gtyp_HBW".History[#li_Counter].i_code := 0;
	                    "gtyp_HBW".History[#li_Counter].ldt_ts := DT#1990-01-01-00:00:00;
	                END_FOR;
	                "gtyp_HBW".x_HBW_Container_Available := FALSE;
	                "gtyp_HBW".x_HBW_PickedUp_Accepted := TRUE;

	                "gtyp_Interface_Dashboard".Subscribe.State_HBW.x_active := FALSE;

	                #li_Lights := 2;
	                #li_StepCase := 190;
	            // VGR discard - storage
	            ELSIF "gtyp_VGR".x_HBW_Discards AND "gtyp_VGR".x_HBW_Storage THEN
	                "gtyp_Interface_Dashboard".Subscribe.State_HBW.x_active := TRUE;
	                "gtyp_HBW".Workpiece := "gtyp_VGR".Workpiece;
	                "gtyp_HBW".History:= "gtyp_VGR".History;
	                "gtyp_HBW".x_HBW_Container_Available := FALSE;
	                "gtyp_HBW".x_HBW_Discards_Accepted := TRUE;
	                #lx_Storage := true;

	                #li_Lights := 2;
	                #li_StepCase := 190;
	            END_IF;

	        190: // Start Conveyor Belt Back

	            IF NOT "gtyp_VGR".x_HBW_Discards AND NOT "gtyp_VGR".x_HBW_PickedUp THEN
	                "QX_HBW_M1_ConveyorBeltBackward_Q2" := TRUE;
	                "QX_HBW_M1_ConveyorBeltForward_Q1" := FALSE;
	                #li_StepCase := 200;
	            END_IF;

	        200:  // Conveyor Belt inside reached

	            #lx_Time_Error := TRUE;

	            IF NOT "IX_HBW_LightBarrierInside_I2" THEN
	                "QX_HBW_M1_ConveyorBeltBackward_Q2" := FALSE;
	                "QX_HBW_M1_ConveyorBeltForward_Q1"  := FALSE;
	                #lx_Time_Error                      := FALSE;
	                #li_StepCase                        := 210;
	            END_IF;

	            // runtime error
	            IF #lfb_TON_Error.Q THEN
	                #li_Lights := 4;
	                #lx_Time_Error := FALSE;
	                "QX_HBW_M1_ConveyorBeltBackward_Q2" := FALSE;
	                "QX_HBW_M1_ConveyorBeltForward_Q1" := FALSE;
	                "gtyp_Interface_Dashboard".Subscribe.State_HBW.x_active := FALSE;
	                "gtyp_HBW".x_Error := TRUE;
	                #li_StepCase := 0;
	            END_IF;

	        210: // Position vertical+offset Belt

	            "gtyp_HBW".Vertical_Axis.di_Target_Position := "gtyp_HBW".di_PosBelt_Vertical - "gtyp_HBW".di_Offset_Pos_Belt_Vertical;
	            "gtyp_HBW".Vertical_Axis.x_Start_Positioning := TRUE;

	            IF ("gtyp_HBW".Vertical_Axis.di_Actual_Position <= ("gtyp_HBW".di_PosBelt_Vertical - "gtyp_HBW".di_Offset_Pos_Belt_Vertical + "gtyp_HBW".Vertical_Axis.Config.di_Pos_Window))
	                AND ("gtyp_HBW".Vertical_Axis.di_Actual_Position >= ("gtyp_HBW".di_PosBelt_Vertical - "gtyp_HBW".di_Offset_Pos_Belt_Vertical - "gtyp_HBW".Vertical_Axis.Config.di_Pos_Window))
	                AND "gtyp_HBW".Vertical_Axis.x_Position_Reached THEN
	                "gtyp_HBW".Vertical_Axis.x_Start_Positioning := FALSE;
	            END_IF;

	            IF ("gtyp_HBW".Vertical_Axis.di_Actual_Position <= ("gtyp_HBW".di_PosBelt_Vertical - "gtyp_HBW".di_Offset_Pos_Belt_Vertical + "gtyp_HBW".Vertical_Axis.Config.di_Pos_Window))
	                AND ("gtyp_HBW".Vertical_Axis.di_Actual_Position >= ("gtyp_HBW".di_PosBelt_Vertical - "gtyp_HBW".di_Offset_Pos_Belt_Vertical - "gtyp_HBW".Vertical_Axis.Config.di_Pos_Window))
	                AND "gtyp_HBW".Vertical_Axis.x_Position_Reached THEN
	                "gtyp_HBW".Vertical_Axis.x_Start_Positioning := FALSE;
	                #li_StepCase := 220;
	            END_IF;

	        220: // Position Cantilever back Belt
	            "QX_HBW_M4_CantileverBackward_Q8" := TRUE;
	            "QX_HBW_M4_CantileverForward_Q7" := FALSE;

	            IF NOT "IX_HBW_SwitchCantileverFront_I5" AND "IX_HBW_SwitchCantileverBack_I6" THEN
	                "QX_HBW_M4_CantileverBackward_Q8" := FALSE;
	                "QX_HBW_M4_CantileverForward_Q7" := FALSE;
	                #li_StepCase := 230;
	            END_IF;

	        230: // Position vertical+offset/horizontal HBW
	            "gtyp_HBW".Horizontal_Axis.di_Target_Position := #ldi_PosRack_Horizontal;
	            "gtyp_HBW".Horizontal_Axis.x_Start_Positioning := TRUE;
	            "gtyp_HBW".Vertical_Axis.di_Target_Position := #ldi_PosRack_Vertical - "gtyp_HBW".di_Offset_Pos_Rack_Vertical;
	            "gtyp_HBW".Vertical_Axis.x_Start_Positioning := TRUE;

	            IF ("gtyp_HBW".Horizontal_Axis.di_Actual_Position <= (#ldi_PosRack_Horizontal + "gtyp_HBW".Horizontal_Axis.Config.di_Pos_Window))
	                AND ("gtyp_HBW".Horizontal_Axis.di_Actual_Position >= (#ldi_PosRack_Horizontal - "gtyp_HBW".Horizontal_Axis.Config.di_Pos_Window))
	                AND "gtyp_HBW".Horizontal_Axis.x_Position_Reached THEN
	                "gtyp_HBW".Horizontal_Axis.x_Start_Positioning := FALSE;
	            END_IF;

	            IF ("gtyp_HBW".Vertical_Axis.di_Actual_Position <= (#ldi_PosRack_Vertical - "gtyp_HBW".di_Offset_Pos_Rack_Vertical + "gtyp_HBW".Vertical_Axis.Config.di_Pos_Window))
	                AND ("gtyp_HBW".Vertical_Axis.di_Actual_Position >= (#ldi_PosRack_Vertical - "gtyp_HBW".di_Offset_Pos_Rack_Vertical - "gtyp_HBW".Vertical_Axis.Config.di_Pos_Window))
	                AND "gtyp_HBW".Vertical_Axis.x_Position_Reached THEN
	                "gtyp_HBW".Vertical_Axis.x_Start_Positioning := FALSE;
	            END_IF;

	            IF ("gtyp_HBW".Horizontal_Axis.di_Actual_Position <= (#ldi_PosRack_Horizontal + "gtyp_HBW".Horizontal_Axis.Config.di_Pos_Window))
	                AND ("gtyp_HBW".Horizontal_Axis.di_Actual_Position >= (#ldi_PosRack_Horizontal - "gtyp_HBW".Horizontal_Axis.Config.di_Pos_Window))
	                AND "gtyp_HBW".Horizontal_Axis.x_Position_Reached
	                AND ("gtyp_HBW".Vertical_Axis.di_Actual_Position <= (#ldi_PosRack_Vertical - "gtyp_HBW".di_Offset_Pos_Rack_Vertical + "gtyp_HBW".Vertical_Axis.Config.di_Pos_Window))
	                AND ("gtyp_HBW".Vertical_Axis.di_Actual_Position >= (#ldi_PosRack_Vertical - "gtyp_HBW".di_Offset_Pos_Rack_Vertical - "gtyp_HBW".Vertical_Axis.Config.di_Pos_Window))
	                AND "gtyp_HBW".Vertical_Axis.x_Position_Reached THEN
	                "gtyp_HBW".Horizontal_Axis.x_Start_Positioning := FALSE;
	                "gtyp_HBW".Vertical_Axis.x_Start_Positioning := FALSE;
	                #li_StepCase := 240;
	            END_IF;

	        240: // Position Cantilever Forward HBW

	            "QX_HBW_M4_CantileverBackward_Q8" := FALSE;
	            "QX_HBW_M4_CantileverForward_Q7" := TRUE;

	            IF "IX_HBW_SwitchCantileverFront_I5" AND NOT "IX_HBW_SwitchCantileverBack_I6" THEN
	                "QX_HBW_M4_CantileverBackward_Q8" := FALSE;
	                "QX_HBW_M4_CantileverForward_Q7" := FALSE;
	                #li_StepCase := 250;
	            END_IF;

	        250: // Position vertical HBW
	            "gtyp_HBW".Vertical_Axis.di_Target_Position := #ldi_PosRack_Vertical;
	            "gtyp_HBW".Vertical_Axis.x_Start_Positioning := TRUE;

	            IF ("gtyp_HBW".Vertical_Axis.di_Actual_Position <= (#ldi_PosRack_Vertical + "gtyp_HBW".Vertical_Axis.Config.di_Pos_Window))
	                AND ("gtyp_HBW".Vertical_Axis.di_Actual_Position >= (#ldi_PosRack_Vertical - "gtyp_HBW".Vertical_Axis.Config.di_Pos_Window))
	                AND "gtyp_HBW".Vertical_Axis.x_Position_Reached THEN
	                IF #lx_Storage THEN
	                    #li_Return_LDT := RD_SYS_T(#ldt_MQTT);
	                    "gtyp_HBW".History[3].i_code := 300;
	                    "gtyp_HBW".History[3].ldt_ts := DT_TO_LDT(#ldt_MQTT);
	                    "gtyp_HBW".Rack_Workpiece[#li_Counter_Act_Ver, #li_Counter_Act_Hor] := "gtyp_HBW".Workpiece;
	                    "gtyp_HBW".Rack_History[#li_Counter_Act_Ver, #li_Counter_Act_Hor].History := "gtyp_HBW".History;
	                    "gtyp_Interface_Dashboard".Subscribe.State_HBW.x_active := FALSE;
	                ELSE
	                    "gtyp_HBW".Rack_Workpiece[#li_Counter_Act_Ver, #li_Counter_Act_Hor].s_id := '0';
	                END_IF;
	                "gtyp_HBW".Vertical_Axis.x_Start_Positioning := FALSE;
	                #li_StepCase := 260;
	            END_IF;

	        260: // Position Cantilever Backward HBW

	            "QX_HBW_M4_CantileverBackward_Q8" := TRUE;
	            "QX_HBW_M4_CantileverForward_Q7" := FALSE;

	            IF NOT "IX_HBW_SwitchCantileverFront_I5" AND "IX_HBW_SwitchCantileverBack_I6" THEN
	                "QX_HBW_M4_CantileverBackward_Q8" := FALSE;
	                "QX_HBW_M4_CantileverForward_Q7" := FALSE;
	                #li_StepCase := 0;
	                #lx_Storage := FALSE;
	            END_IF;
	    // Statement section ELSE
	    ELSE
	        ;
	    END_CASE;

	    //Reset the information in the high-bay warehouse
	    IF "gtyp_Setup".x_Clean_Rack_HBW THEN
	        FOR #li_Counter_Hor := 1 TO 3 DO
	            FOR #li_Counter_Ver := 1 TO 3 DO
	                "gtyp_HBW".Rack_Workpiece[#li_Counter_Ver, #li_Counter_Hor].s_id := '0';
	                "gtyp_HBW".Rack_Workpiece[#li_Counter_Ver, #li_Counter_Hor].s_state := '';
	                "gtyp_HBW".Rack_Workpiece[#li_Counter_Ver, #li_Counter_Hor].s_type := '';
	                FOR #li_Counter := 1 TO 8 DO
	                    "gtyp_HBW".Rack_History[#li_Counter_Ver, #li_Counter_Hor].History[#li_Counter].i_code := 0;
	                    "gtyp_HBW".Rack_History[#li_Counter_Ver, #li_Counter_Hor].History[#li_Counter].ldt_ts := DT#1990-01-01-00:00:00;
	                END_FOR;
	            END_FOR;
	        END_FOR;
	        "gtyp_Setup".x_Clean_Rack_HBW := FALSE;
	    END_IF;

	    // reload PWM
	    "QW_HBW_PWM_ConveyorBelt_M1"   := "gtyp_HBW"."i_PWM_ConveyorBelt";
	    "QW_HBW_PWM_Cantilever_M4"     := "gtyp_HBW"."i_PWM_Cantilever";
	ELSE
	    FOR #li_Counter_Hor := 1 TO 3 DO
	        FOR #li_Counter_Ver := 1 TO 3 DO
	            IF "gtyp_HBW".Rack_Workpiece[#li_Counter_Ver, #li_Counter_Hor].s_id = '' THEN
	                "gtyp_HBW".Rack_Workpiece[#li_Counter_Ver, #li_Counter_Hor].s_id := '0';
	                "gtyp_HBW".Rack_Workpiece[#li_Counter_Ver, #li_Counter_Hor].s_state := '';
	                "gtyp_HBW".Rack_Workpiece[#li_Counter_Ver, #li_Counter_Hor].s_type := '';
	                FOR #li_Counter := 1 TO 8 DO
	                    "gtyp_HBW".Rack_History[#li_Counter_Ver, #li_Counter_Hor].History[#li_Counter].i_code := 0;
	                    "gtyp_HBW".Rack_History[#li_Counter_Ver, #li_Counter_Hor].History[#li_Counter].ldt_ts := DT#1990-01-01-00:00:00;
	                END_FOR;
	            END_IF;
	        END_FOR;
	    END_FOR;

	    "gtyp_HBW".x_Start_Park_Position := FALSE;
	    "gtyp_HBW".x_Park_Position_Reached := FALSE;
	    "gtyp_HBW".x_HBW_PickedUp_Accepted := FALSE;
	    "gtyp_HBW".x_HBW_Discards_Accepted := FALSE;
	    "gtyp_HBW".x_HBW_PickUp_Ready := FALSE;
	    "gtyp_HBW".x_HBW_Container_Available := FALSE;
	    "gtyp_HBW".x_Error := FALSE;

	    #li_Lights := 1;
	    #lx_Init := TRUE;
	END_IF;
END_FUNCTION_BLOCK

FUNCTION_BLOCK "PRG_VGR_Axis_rotate"
TITLE = Program Axis rotate VGR
{ S7_Optimized_Access := 'TRUE' }
AUTHOR : 'A.Schaefer'
VERSION : 0.0
   VAR
      lx_Init { ExternalAccessible := 'False'; ExternalVisible := 'False'; ExternalWritable := 'False'} : Bool;
      lfb_rotate_Axis { ExternalAccessible := 'False'; ExternalVisible := 'False'; ExternalWritable := 'False'; S7_SetPoint := 'False'} : "FB_Axis";
   END_VAR


BEGIN
	IF #lx_Init THEN

	    // FB Axis rotate
	    #lfb_rotate_Axis(ini_Axis           := 3,
	                indi_Increment          := "gtyp_VGR".rotate_Axis.di_Increment,
	                inx_Ref_Switch          := "IX_VGR_RefSwitchRotate_I3",
	                inx_Referencing         := "gtyp_VGR".rotate_Axis.x_Reference,
	                inx_Start_Positioning   := "gtyp_VGR".rotate_Axis.x_Start_Positioning,
	                indi_Target_Position    := "gtyp_VGR".rotate_Axis.di_Target_Position,
	                ini_PWM                 := "gtyp_VGR".rotate_Axis.i_PWM,
	                inouttyp_Config         := "gtyp_VGR".rotate_Axis.Config,
	                inouttyp_Setup          := "gtyp_SetupAxis");

	    "QX_VGR_M3_RotateClockwise_Q5"          := #lfb_rotate_Axis.outx_Motor_Neg;
	    "QX_VGR_M3_RotateCounterclockwise_Q6"   := #lfb_rotate_Axis.outx_Motor_Pos;
	    "QW_VGR_PWM_Rotate_M3"                  := #lfb_rotate_Axis.outi_Motor_PWM;
	    "gtyp_VGR".rotate_Axis.di_Actual_Position := #lfb_rotate_Axis.outdi_Actual_Position;
	    "gtyp_VGR".rotate_Axis.x_Referenced       := #lfb_rotate_Axis.outx_Referenced;
	    "gtyp_VGR".rotate_Axis.x_Position_Reached := #lfb_rotate_Axis.outx_Position_Reached;
	ELSE
	    #lx_Init := TRUE;
	END_IF;
END_FUNCTION_BLOCK

FUNCTION_BLOCK "PRG_SSC_Calibration_Color"
TITLE = Program Calibration Color Sensor SSC
{ S7_Optimized_Access := 'TRUE' }
AUTHOR : 'A.Schaefer'
VERSION : 0.0
   VAR
      lx_Init { ExternalAccessible := 'False'; ExternalVisible := 'False'; ExternalWritable := 'False'} : Bool;
      lx_Start_TON_Wait { ExternalAccessible := 'False'; ExternalVisible := 'False'; ExternalWritable := 'False'} : Bool;
      lx_Start_Positioning_m { ExternalAccessible := 'False'; ExternalVisible := 'False'; ExternalWritable := 'False'} : Bool;
      lt_TON_Wait { ExternalAccessible := 'False'; ExternalVisible := 'False'; ExternalWritable := 'False'} : Time;
      li_StepCase { ExternalAccessible := 'False'; ExternalVisible := 'False'; ExternalWritable := 'False'} : Int;
      ldi_Pos_Horizontal { ExternalAccessible := 'False'; ExternalVisible := 'False'; ExternalWritable := 'False'} : DInt;
      ldi_Pos_Vertical { ExternalAccessible := 'False'; ExternalVisible := 'False'; ExternalWritable := 'False'} : DInt;
      lfb_R_Trig_Deaktivate {InstructionName := 'R_TRIG'; LibVersion := '1.0'; ExternalAccessible := 'False'; ExternalVisible := 'False'; ExternalWritable := 'False'; S7_SetPoint := 'False'} : R_TRIG;
      lfb_TON_Wait {InstructionName := 'TON_TIME'; LibVersion := '1.0'; ExternalAccessible := 'False'; ExternalVisible := 'False'; ExternalWritable := 'False'; S7_SetPoint := 'False'} : TON_TIME;
   END_VAR


BEGIN
	IF #lx_Init THEN

	    // FB TON Wait
	    #lfb_TON_Wait(IN := #lx_Start_TON_Wait,
	                  PT := #lt_TON_Wait);

	    #lfb_R_Trig_Deaktivate(CLK:= NOT "gtyp_Setup".x_Color_Sensor_Calibration
	                           OR NOT ("gtyp_Setup".i_Color_Sensor_Selection = 1));
	    // Deaktivate step 0
	    IF #lfb_R_Trig_Deaktivate.Q THEN
	        "gtyp_Setup".x_Calculate_Value_Color := FALSE;
	        "gtyp_Setup".x_Set_Calib_Value_Color_Blue := FALSE;
	        "gtyp_Setup".x_Set_Calib_Value_Color_Red := FALSE;
	        "gtyp_Setup".x_Set_Calib_Value_Color_White := FALSE;
	        "gtyp_Setup".w_Calib_ColorValue_Blue := 0;
	        "gtyp_Setup".w_Calib_ColorValue_Red := 0;
	        "gtyp_Setup".w_Calib_ColorValue_White := 0;
	        "gtyp_Setup".w_Threshold_Red_Blue := 0;
	        "gtyp_Setup".w_Threshold_White_Red := 0;
	        #li_StepCase            := 0;
	    END_IF;

	    // step chain HBW
	    CASE #li_StepCase OF

	        0:  // init
	            #lx_Start_TON_Wait := FALSE;
	            #li_StepCase := 10;

	        10:  // Set Calibration activ?
	            IF "gtyp_Setup".x_Color_Sensor_Calibration
	                AND ("gtyp_Setup".i_Color_Sensor_Selection = 1) THEN
	                "gtyp_Setup".x_Calculate_Value_Color := FALSE;
	                "gtyp_Setup".x_Set_Calib_Value_Color_Blue := FALSE;
	                "gtyp_Setup".x_Set_Calib_Value_Color_Red := FALSE;
	                "gtyp_Setup".x_Set_Calib_Value_Color_White := FALSE;
	                "gtyp_Setup".w_Calib_ColorValue_Blue := 0;
	                "gtyp_Setup".w_Calib_ColorValue_Red := 0;
	                "gtyp_Setup".w_Calib_ColorValue_White := 0;
	                "gtyp_Setup".w_Threshold_Red_Blue := 0;
	                "gtyp_Setup".w_Threshold_White_Red := 0;
	                #li_StepCase := 20;
	            END_IF;

	        20: // wait for set Values or Calculate

	            // Start new Positioning
	            IF "gtyp_Setup".x_Set_Calib_Value_Color_Blue THEN
	                "gtyp_Setup".w_Calib_ColorValue_Blue := "IW_SSC_ColorSensor_A1";
	                "gtyp_Setup".x_Set_Calib_Value_Color_Blue := FALSE;
	            ELSIF "gtyp_Setup".x_Set_Calib_Value_Color_Red THEN
	                "gtyp_Setup".w_Calib_ColorValue_Red := "IW_SSC_ColorSensor_A1";
	                "gtyp_Setup".x_Set_Calib_Value_Color_Red := FALSE;
	            ELSIF "gtyp_Setup".x_Set_Calib_Value_Color_White THEN
	                "gtyp_Setup".w_Calib_ColorValue_White := "IW_SSC_ColorSensor_A1";
	                "gtyp_Setup".x_Set_Calib_Value_Color_White := FALSE;
	            END_IF;

	            "gtyp_Setup".w_Threshold_White_Red  := "gtyp_Setup".w_Calib_ColorValue_White + (("gtyp_Setup".w_Calib_ColorValue_Red - "gtyp_Setup".w_Calib_ColorValue_White) / 2);
	            "gtyp_Setup".w_Threshold_Red_Blue   := "gtyp_Setup".w_Calib_ColorValue_Red + (("gtyp_Setup".w_Calib_ColorValue_Blue - "gtyp_Setup".w_Calib_ColorValue_Red) / 2);

	            IF "gtyp_Setup".x_Calculate_Value_Color THEN
	                "gtyp_SSC".w_Threshold_White_Red := "gtyp_Setup".w_Threshold_White_Red;
	                "gtyp_SSC".w_Threshold_Red_Blue := "gtyp_Setup".w_Threshold_Red_Blue;
	                "gtyp_Setup".x_Calculate_Value_Color := FALSE;
	            END_IF;

	            // Statement section ELSE
	        ELSE
	            ;
	    END_CASE;

	    IF ("gtyp_Setup".i_Color_Sensor_Selection = 1) THEN
	        // Reload Pos Value
	        "gtyp_Setup".w_Actual_ColorValue := "IW_SSC_ColorSensor_A1";
	    END_IF;
	ELSE
	    #lx_Init := TRUE;
	END_IF;
END_FUNCTION_BLOCK

FUNCTION_BLOCK "PRG_VGR_Axis_horizontal"
TITLE = Program Axis horizontal VGR
{ S7_Optimized_Access := 'TRUE' }
AUTHOR : 'A.Schaefer'
VERSION : 0.0
   VAR
      lx_Init { ExternalAccessible := 'False'; ExternalVisible := 'False'; ExternalWritable := 'False'} : Bool;
      lfb_horizontal_Axis { ExternalAccessible := 'False'; ExternalVisible := 'False'; ExternalWritable := 'False'; S7_SetPoint := 'False'} : "FB_Axis";
   END_VAR


BEGIN
	IF #lx_Init THEN

	    // FB Axis horizontal
	    #lfb_horizontal_Axis(ini_Axis       := 1,
	                indi_Increment          := "gtyp_VGR".horizontal_Axis.di_Increment,
	                inx_Ref_Switch          := "IX_VGR_RefSwitchHorizontalAxis_I2",
	                inx_Referencing         := "gtyp_VGR".horizontal_Axis.x_Reference,
	                inx_Start_Positioning   := "gtyp_VGR".horizontal_Axis.x_Start_Positioning,
	                indi_Target_Position    := "gtyp_VGR".horizontal_Axis.di_Target_Position,
	                ini_PWM                 := "gtyp_VGR".horizontal_Axis.i_PWM,
	                inouttyp_Config         := "gtyp_VGR".horizontal_Axis.Config,
	                inouttyp_Setup          := "gtyp_SetupAxis");

	    "QX_VGR_M2_HorizontalAxisForward_Q4"    := #lfb_horizontal_Axis.outx_Motor_Pos;
	    "QX_VGR_M2_HorizontalAxisBackward_Q3"   := #lfb_horizontal_Axis.outx_Motor_Neg;
	    "QW_VGR_PWM_Horizontal_M2"              := #lfb_horizontal_Axis.outi_Motor_PWM;
	    "gtyp_VGR".horizontal_Axis.di_Actual_Position    := #lfb_horizontal_Axis.outdi_Actual_Position;
	    "gtyp_VGR".horizontal_Axis.x_Referenced          := #lfb_horizontal_Axis.outx_Referenced;
	    "gtyp_VGR".horizontal_Axis.x_Position_Reached    := #lfb_horizontal_Axis.outx_Position_Reached;
	ELSE
	    #lx_Init := TRUE;
	END_IF;
END_FUNCTION_BLOCK

FUNCTION_BLOCK "PRG_MPO_Ablauf"
TITLE = Program Ablauf MPO
{ S7_Optimized_Access := 'TRUE' }
AUTHOR : 'A.Schaefer'
VERSION : 0.0
   VAR
      lx_Init { ExternalAccessible := 'False'; ExternalVisible := 'False'; ExternalWritable := 'False'} : Bool;
      lx_Start_TON_Wait { ExternalAccessible := 'False'; ExternalVisible := 'False'; ExternalWritable := 'False'} : Bool;
      lx_Time_Error { ExternalAccessible := 'False'; ExternalVisible := 'False'; ExternalWritable := 'False'} : Bool;
      lt_TON_Wait { ExternalAccessible := 'False'; ExternalVisible := 'False'; ExternalWritable := 'False'} : Time;
      lx_Start_TON_State { ExternalAccessible := 'False'; ExternalVisible := 'False'; ExternalWritable := 'False'} : Bool;
      ldt_MQTT { ExternalAccessible := 'False'; ExternalVisible := 'False'; ExternalWritable := 'False'} : Date_And_Time;
      li_Return_LDT { ExternalAccessible := 'False'; ExternalVisible := 'False'; ExternalWritable := 'False'} : Int;
      li_StepCase { ExternalAccessible := 'False'; ExternalVisible := 'False'; ExternalWritable := 'False'} : Int;
      li_Lights { ExternalAccessible := 'False'; ExternalVisible := 'False'; ExternalWritable := 'False'} : Int;
      li_Lights_old { ExternalAccessible := 'False'; ExternalVisible := 'False'; ExternalWritable := 'False'} : Int;
      li_Counter { ExternalAccessible := 'False'; ExternalVisible := 'False'; ExternalWritable := 'False'} : Int;
      lfb_blinker { ExternalAccessible := 'False'; ExternalVisible := 'False'; ExternalWritable := 'False'; S7_SetPoint := 'False'} : "FB_Blinker";
      lfb_TOF_ConveyerBelt_Out {InstructionName := 'TOF_TIME'; LibVersion := '1.0'; ExternalAccessible := 'False'; ExternalVisible := 'False'; ExternalWritable := 'False'; S7_SetPoint := 'False'} : TOF_TIME;
      lfb_TON_Wait {InstructionName := 'TON_TIME'; LibVersion := '1.0'; ExternalAccessible := 'False'; ExternalVisible := 'False'; ExternalWritable := 'False'; S7_SetPoint := 'False'} : TON_TIME;
      lfb_TON_Error {InstructionName := 'TON_TIME'; LibVersion := '1.0'; ExternalAccessible := 'False'; ExternalVisible := 'False'; ExternalWritable := 'False'; S7_SetPoint := 'False'} : TON_TIME;
      lfb_TON_State {InstructionName := 'TON_TIME'; LibVersion := '1.0'; ExternalAccessible := 'False'; ExternalVisible := 'False'; ExternalWritable := 'False'; S7_SetPoint := 'False'} : TON_TIME;
      lfb_F_Trig_ConveyerBelt {InstructionName := 'F_TRIG'; LibVersion := '1.0'; ExternalAccessible := 'False'; ExternalVisible := 'False'; ExternalWritable := 'False'; S7_SetPoint := 'False'} : F_TRIG;
   END_VAR


BEGIN
	IF #lx_Init THEN

	    // wait time state
	    #lfb_TON_State(IN := NOT #lx_Start_TON_State,
	                    PT := T#2s);

	    // runtime monitoring error
	    #lfb_TON_Error(IN := #lx_Time_Error,
	                   PT := T#30s);

	    // state of the MPO cyclically transmitted to the cloud
	    IF (#lfb_TON_State.Q OR (#li_Lights <> #li_Lights_old)) AND NOT #lx_Start_TON_State THEN
	        #li_Lights_old := #li_Lights;
	        #lx_Start_TON_State := TRUE;
	        #li_Return_LDT := RD_SYS_T(#ldt_MQTT);
	        "gtyp_Interface_Dashboard".Subscribe.State_MPO.ldt_ts        := DT_TO_LDT(#ldt_MQTT);
	        "gtyp_Interface_Dashboard".Subscribe.State_MPO.i_code        := #li_Lights;
	        "gtyp_Interface_Dashboard".Subscribe.State_MPO.s_description := '';
	        "gtyp_Interface_Dashboard".Subscribe.State_MPO.s_station     := 'mpo';
	        "gtyp_Interface_Dashboard".Subscribe.State_MPO.s_target      := '';
	    END_IF;

	    // restart wait time state
	    IF NOT #lfb_TON_State.Q AND #lx_Start_TON_State THEN
	        #lx_Start_TON_State := FALSE;
	    END_IF;

	    // FB TON Wait
	    #lfb_TON_Wait(IN := #lx_Start_TON_Wait,
	                    PT := #lt_TON_Wait);

	   // falling edge light barrier end of Conveyor Belt
	   #lfb_F_Trig_ConveyerBelt(CLK := NOT "IX_MPO_LightBarrierEndOfConBelt_I3");

	    //Run-on time Conveyer Belt
	   #lfb_TOF_ConveyerBelt_Out(IN:= #lfb_F_Trig_ConveyerBelt.Q,
	                             PT:= T#5000ms);

	    // FB blinker intervall 1s
	    #lfb_blinker(int_periodendauer:= T#1000ms);

	    // step chain HBW
	    CASE #li_StepCase OF

	        0:  // init
	            #lx_Start_TON_Wait := FALSE;
	            #lx_Time_Error := FALSE;

	            IF NOT "gtyp_MPO".x_Error AND NOT "gtyp_MPO".x_Start_Park_Position THEN
	                #li_StepCase := 10;
	            END_IF;

	        10: // turn-on Compressor and turn off oven light
	            #li_Lights := 2;
	            "QX_MPO_LightOven_Q9"   := FALSE;
	            "QX_MPO_Compressor_Q10" := TRUE;

	            #lx_Start_TON_Wait := TRUE;
	            #lt_TON_Wait := T#500ms;

	            IF #lfb_TON_Wait.Q THEN
	                #lx_Start_TON_Wait := FALSE;
	                #li_StepCase := 20;
	            END_IF;

	        20:  // Open oven door
	            "QX_MPO_ValveOvenDoor_Q13" := TRUE;
	            "QX_MPO_ValveLowering_Q12" := FALSE;

	            #lx_Start_TON_Wait := TRUE;
	            #lt_TON_Wait := T#2000ms;

	            IF #lfb_TON_Wait.Q THEN
	                #lx_Start_TON_Wait := FALSE;
	                #li_StepCase := 30;
	            END_IF;

	        30: // Position oven feeder retract
	            IF "IX_MPO_RefSwitchOvenFeederOutside_I7" OR NOT "IX_MPO_RefSwitchOvenFeederInside_I6" THEN
	                "QX_MPO_M4_OvenFeederRetract_Q5" := TRUE;
	                "QX_MPO_M4_OvenFeederExtend_Q6" := FALSE;
	            ELSIF NOT "IX_MPO_RefSwitchOvenFeederOutside_I7" AND "IX_MPO_RefSwitchOvenFeederInside_I6" THEN
	                "QX_MPO_M4_OvenFeederRetract_Q5" := FALSE;
	                "QX_MPO_M4_OvenFeederExtend_Q6" := FALSE;
	                #li_StepCase := 40;
	            END_IF;

	        40:  // Close door, Position Vacuum Towards Turn Table and vacuum off

	            "QX_MPO_ValveOvenDoor_Q13" := FALSE;

	            "QX_MPO_M5_VacuumTowardsTurnTable_Q8" := TRUE;
	            "QX_MPO_M5_VacuumTowardsOven_Q7" := FALSE;
	            "QX_MPO_ValveVacuum_Q11"        := FALSE;

	            IF"IX_MPO_RefSwitchVac_PosOven_I8" OR NOT "IX_MPO_RefSwitchVac_PosTurnTable_I5" THEN
	                "QX_MPO_M5_VacuumTowardsTurnTable_Q8" := TRUE;
	                "QX_MPO_M5_VacuumTowardsOven_Q7" := FALSE;
	            ELSIF NOT "IX_MPO_RefSwitchVac_PosOven_I8" AND "IX_MPO_RefSwitchVac_PosTurnTable_I5" THEN
	                "QX_MPO_M5_VacuumTowardsTurnTable_Q8" := FALSE;
	                "QX_MPO_M5_VacuumTowardsOven_Q7" := FALSE;
	                #li_StepCase := 50;
	            END_IF
	            ;

	        50: // saw, valve feeder conveyor belt off
	            "QX_MPO_M3_Saw_Q4" := FALSE;
	            "QX_MPO_ValveFeeder_Q14" := FALSE;
	            "QX_MPO_M2_ConveyorBeltForward_Q3" := FALSE;

	            IF "IX_MPO_RefSwitchTurnTable_PosSaw_I4" OR "IX_MPO_RefSwitchTurnTable_PosBelt_I2" OR NOT "IX_MPO_RefSwitchTurnTable_PosVac_I1" THEN
	                "QX_MPO_M1_TurnTableClockwise_Q1" := FALSE;
	                "QX_MPO_M1_TurnTableCounterclockwise_Q2" := TRUE;
	            ELSIF NOT "IX_MPO_RefSwitchTurnTable_PosSaw_I4" AND NOT "IX_MPO_RefSwitchTurnTable_PosBelt_I2" AND "IX_MPO_RefSwitchTurnTable_PosVac_I1" THEN
	                "QX_MPO_M1_TurnTableClockwise_Q1" := FALSE;
	                "QX_MPO_M1_TurnTableCounterclockwise_Q2" := FALSE;
	                "QX_MPO_Compressor_Q10" := FALSE;
	                #li_StepCase := 60;
	            END_IF;

	        60: // wait for request discard form VGR
	            #li_Lights := 1;
	            IF "gtyp_VGR".x_MPO_Req_Discard THEN
	                #li_Lights := 2;
	                "QX_MPO_Compressor_Q10" := TRUE;
	                #li_StepCase := 70;
	            END_IF;

	        70: // wait sequence
	            #lx_Start_TON_Wait := TRUE;
	            #lt_TON_Wait := T#500ms;

	            IF #lfb_TON_Wait.Q THEN
	                #lx_Start_TON_Wait := FALSE;
	                #li_StepCase := 80;
	            END_IF;

	        80: // open oven door
	            "QX_MPO_ValveOvenDoor_Q13" := TRUE;

	            #lx_Start_TON_Wait := TRUE;
	            #lt_TON_Wait := T#2000ms;

	            IF #lfb_TON_Wait.Q THEN
	                #lx_Start_TON_Wait := FALSE;
	                #li_StepCase := 90;
	            END_IF;

	        90: // oven feeder extend
	            "QX_MPO_M4_OvenFeederRetract_Q5"    := FALSE;
	            "QX_MPO_M4_OvenFeederExtend_Q6"     := TRUE;

	            IF "IX_MPO_RefSwitchOvenFeederOutside_I7" AND NOT "IX_MPO_RefSwitchOvenFeederInside_I6" THEN
	                "QX_MPO_M4_OvenFeederRetract_Q5" := FALSE;
	                "QX_MPO_M4_OvenFeederExtend_Q6" := FALSE;
	                "gtyp_MPO".x_MPO_Discards_Accepted := FALSE;
	                "gtyp_MPO".x_Discard_Ready      := TRUE;
	                #li_StepCase := 100;
	            END_IF;

	        100: // wait for VGR discard workpiece

	            #lx_Time_Error := TRUE;

	            IF "gtyp_VGR".x_MPO_Discards AND NOT "IX_MPO_LightBarrierOven_I9" THEN
	                "gtyp_Interface_Dashboard".Subscribe.State_MPO.x_active := TRUE;
	                "gtyp_MPO".History  := "gtyp_VGR".History;
	                "gtyp_MPO".Workpiece := "gtyp_VGR".Workpiece;
	                "gtyp_MPO".x_Discard_Ready := FALSE;
	                "gtyp_MPO".x_MPO_Discards_Accepted := TRUE;
	                #lx_Time_Error := FALSE;
	                #li_StepCase := 105;
	            END_IF;

	            // runtime error
	            IF #lfb_TON_Error.Q THEN
	                #li_Lights := 4;
	                #lx_Time_Error := FALSE;
	                "gtyp_Interface_Dashboard".Subscribe.State_Order.ldt_ts := DT_TO_LDT(#ldt_MQTT);
	                "gtyp_Interface_Dashboard".Subscribe.State_Order.s_state := 'WAITING_FOR_ORDER';
	                "gtyp_Interface_Dashboard".Subscribe.State_Order.s_type := '';
	                "gtyp_Interface_Dashboard".Subscribe.State_MPO.x_active := FALSE;
	                "gtyp_MPO".x_Discard_Ready := FALSE;
	                "gtyp_MPO".x_MPO_Discards_Accepted := FALSE;
	                "gtyp_MPO".x_Error := TRUE;
	                #li_StepCase := 0;
	            END_IF;

	        105: // VGR outside oven feeder - oven feeder retract
	            IF NOT "gtyp_VGR".x_MPO_Discards AND "IX_MPO_RefSwitchOvenFeederOutside_I7" AND NOT "IX_MPO_RefSwitchOvenFeederInside_I6" THEN
	                "gtyp_MPO".x_MPO_Discards_Accepted := FALSE;
	                "QX_MPO_M4_OvenFeederRetract_Q5" := TRUE;
	                "QX_MPO_M4_OvenFeederExtend_Q6" := FALSE;
	                #li_StepCase := 110;
	            END_IF;

	        110: // sensor oven feeder inside reached
	            IF NOT "IX_MPO_RefSwitchOvenFeederOutside_I7" AND "IX_MPO_RefSwitchOvenFeederInside_I6" THEN
	                "QX_MPO_M4_OvenFeederRetract_Q5" := FALSE;
	                "QX_MPO_M4_OvenFeederExtend_Q6" := FALSE;
	                #li_StepCase := 120;
	            END_IF;

	        120: // close oven door
	            "QX_MPO_ValveOvenDoor_Q13" := FALSE;

	            #lx_Start_TON_Wait := TRUE;
	            #lt_TON_Wait := T#2000ms;

	            IF #lfb_TON_Wait.Q THEN
	                #lx_Start_TON_Wait := FALSE;
	                #li_StepCase := 130;
	            END_IF;

	        130: // processing time flashing interval
	            "QX_MPO_LightOven_Q9":= #lfb_blinker.outx_blinker;

	            IF NOT "gtyp_VGR".x_MPO_Discards THEN
	                #li_Return_LDT := RD_SYS_T(#ldt_MQTT);
	                "gtyp_MPO".History[5].i_code := 500;
	                "gtyp_MPO".History[5].ldt_ts := DT_TO_LDT(#ldt_MQTT);

	                "QX_MPO_M5_VacuumTowardsOven_Q7" := TRUE;
	                "QX_MPO_M5_VacuumTowardsTurnTable_Q8" := FALSE;

	                IF NOT "IX_MPO_RefSwitchVac_PosTurnTable_I5" AND "IX_MPO_RefSwitchVac_PosOven_I8" THEN
	                    "QX_MPO_M5_VacuumTowardsOven_Q7" := FALSE;
	                    "QX_MPO_M5_VacuumTowardsTurnTable_Q8" := FALSE;
	                END_IF;
	            END_IF;

	            #lx_Start_TON_Wait := TRUE;
	            #lt_TON_Wait := T#4000ms;

	            IF #lfb_TON_Wait.Q THEN
	                #lx_Start_TON_Wait := FALSE;
	                #li_StepCase := 140;
	            END_IF;

	        140: // open oven door
	            "QX_MPO_LightOven_Q9"       := FALSE;
	            "QX_MPO_ValveOvenDoor_Q13"  := TRUE;

	            IF NOT "gtyp_VGR".x_MPO_Discards THEN
	                "QX_MPO_M5_VacuumTowardsOven_Q7" := TRUE;
	                "QX_MPO_M5_VacuumTowardsTurnTable_Q8" := FALSE;

	                IF NOT "IX_MPO_RefSwitchVac_PosTurnTable_I5" AND "IX_MPO_RefSwitchVac_PosOven_I8" THEN
	                    "QX_MPO_M5_VacuumTowardsOven_Q7" := FALSE;
	                    "QX_MPO_M5_VacuumTowardsTurnTable_Q8" := FALSE;
	                END_IF;
	            END_IF;

	            #lx_Start_TON_Wait := TRUE;
	            #lt_TON_Wait := T#2000ms;

	            IF #lfb_TON_Wait.Q THEN
	                #lx_Start_TON_Wait := FALSE;
	                #li_StepCase := 150;
	            END_IF;

	        150: // oven feeder extend

	            "QX_MPO_M4_OvenFeederRetract_Q5" := FALSE;
	            "QX_MPO_M4_OvenFeederExtend_Q6" := TRUE;

	            IF NOT "gtyp_VGR".x_MPO_Discards THEN
	                "QX_MPO_M5_VacuumTowardsOven_Q7" := TRUE;
	                "QX_MPO_M5_VacuumTowardsTurnTable_Q8" := FALSE;

	                IF NOT "IX_MPO_RefSwitchVac_PosTurnTable_I5" AND "IX_MPO_RefSwitchVac_PosOven_I8" THEN
	                    "QX_MPO_M5_VacuumTowardsOven_Q7" := FALSE;
	                    "QX_MPO_M5_VacuumTowardsTurnTable_Q8" := FALSE;
	                END_IF;
	            END_IF;

	            IF "IX_MPO_RefSwitchOvenFeederOutside_I7" AND NOT "IX_MPO_RefSwitchOvenFeederInside_I6" THEN
	                "QX_MPO_M4_OvenFeederRetract_Q5" := FALSE;
	                "QX_MPO_M4_OvenFeederExtend_Q6" := FALSE;
	            END_IF;

	            IF "IX_MPO_RefSwitchOvenFeederOutside_I7" AND NOT "IX_MPO_RefSwitchOvenFeederInside_I6"
	                AND NOT "IX_MPO_RefSwitchVac_PosTurnTable_I5" AND "IX_MPO_RefSwitchVac_PosOven_I8" THEN
	                "QX_MPO_M5_VacuumTowardsOven_Q7" := FALSE;
	                "QX_MPO_M5_VacuumTowardsTurnTable_Q8" := FALSE;
	                "QX_MPO_M4_OvenFeederRetract_Q5" := FALSE;
	                "QX_MPO_M4_OvenFeederExtend_Q6" := FALSE;
	                #li_StepCase := 160;
	            END_IF;

	        160: // vacuum suction device down
	            "QX_MPO_ValveLowering_Q12":= TRUE;

	            #lx_Start_TON_Wait := TRUE;
	            #lt_TON_Wait := T#1000ms;

	            IF #lfb_TON_Wait.Q THEN
	                #lx_Start_TON_Wait := FALSE;
	                #li_StepCase := 170;
	            END_IF;

	        170: // vacuum suction device picks up the workpiece
	            "QX_MPO_ValveVacuum_Q11":= TRUE;

	            #lx_Start_TON_Wait := TRUE;
	            #lt_TON_Wait := T#1000ms;

	            IF #lfb_TON_Wait.Q THEN
	                #lx_Start_TON_Wait := FALSE;
	                #li_StepCase := 180;
	            END_IF;

	        180: // vacuum suction device up
	            "QX_MPO_ValveLowering_Q12" := FALSE;

	            #lx_Start_TON_Wait := TRUE;
	            #lt_TON_Wait := T#1000ms;

	            IF #lfb_TON_Wait.Q THEN
	                #lx_Start_TON_Wait := FALSE;
	                #li_StepCase := 190;
	            END_IF;

	        190: // oven feeder retract and vacuum towards turn table
	            "QX_MPO_M4_OvenFeederRetract_Q5" := TRUE;
	            "QX_MPO_M4_OvenFeederExtend_Q6" := FALSE;
	            "QX_MPO_M5_VacuumTowardsOven_Q7" := FALSE;
	            "QX_MPO_M5_VacuumTowardsTurnTable_Q8" := TRUE;

	            IF "IX_MPO_RefSwitchVac_PosTurnTable_I5" AND NOT "IX_MPO_RefSwitchVac_PosOven_I8" THEN
	                "QX_MPO_M5_VacuumTowardsOven_Q7" := FALSE;
	                "QX_MPO_M5_VacuumTowardsTurnTable_Q8" := FALSE;
	            END_IF;

	            IF NOT "IX_MPO_RefSwitchOvenFeederOutside_I7" AND "IX_MPO_RefSwitchOvenFeederInside_I6" THEN
	                "QX_MPO_M4_OvenFeederRetract_Q5" := FALSE;
	                "QX_MPO_M4_OvenFeederExtend_Q6" := FALSE;
	            END_IF;

	            IF NOT "IX_MPO_RefSwitchOvenFeederOutside_I7" AND "IX_MPO_RefSwitchOvenFeederInside_I6"
	                AND "IX_MPO_RefSwitchVac_PosTurnTable_I5" AND NOT "IX_MPO_RefSwitchVac_PosOven_I8" THEN
	                "QX_MPO_M5_VacuumTowardsOven_Q7" := FALSE;
	                "QX_MPO_M5_VacuumTowardsTurnTable_Q8" := FALSE;
	                "QX_MPO_M4_OvenFeederRetract_Q5" := FALSE;
	                "QX_MPO_M4_OvenFeederExtend_Q6" := FALSE;
	                "QX_MPO_ValveOvenDoor_Q13" := FALSE;
	                #li_StepCase := 200;
	            END_IF;

	        200: // vacuum suction device down at turn table
	            IF "IX_MPO_RefSwitchTurnTable_PosVac_I1" THEN
	                "QX_MPO_ValveLowering_Q12" := TRUE;

	                #lx_Start_TON_Wait := TRUE;
	                #lt_TON_Wait := T#2000ms;

	                IF #lfb_TON_Wait.Q THEN
	                    #lx_Start_TON_Wait := FALSE;
	                    #li_StepCase := 210;
	                END_IF;
	            END_IF;

	        210: // vacuum off
	            "QX_MPO_ValveVacuum_Q11" := FALSE;

	            #lx_Start_TON_Wait := TRUE;
	            #lt_TON_Wait := T#2000ms;

	            IF #lfb_TON_Wait.Q THEN
	                #lx_Start_TON_Wait := FALSE;
	                #li_StepCase := 220;
	            END_IF;

	        220: // vacuum suction device up
	            "QX_MPO_ValveLowering_Q12" := FALSE;

	            #lx_Start_TON_Wait := TRUE;
	            #lt_TON_Wait := T#2000ms;

	            IF #lfb_TON_Wait.Q THEN
	                #lx_Start_TON_Wait := FALSE;
	                #li_StepCase := 230;
	            END_IF;

	        230: // Position turn table saw
	            IF NOT "IX_MPO_RefSwitchTurnTable_PosSaw_I4" AND NOT "IX_MPO_RefSwitchTurnTable_PosBelt_I2" AND "IX_MPO_RefSwitchTurnTable_PosVac_I1" THEN
	                "QX_MPO_M1_TurnTableClockwise_Q1" := TRUE;
	                "QX_MPO_M1_TurnTableCounterclockwise_Q2" := FALSE;
	            ELSIF "IX_MPO_RefSwitchTurnTable_PosSaw_I4" OR "IX_MPO_RefSwitchTurnTable_PosBelt_I2" AND NOT "IX_MPO_RefSwitchTurnTable_PosVac_I1" THEN
	                "QX_MPO_M1_TurnTableClockwise_Q1" := FALSE;
	                "QX_MPO_M1_TurnTableCounterclockwise_Q2" := FALSE;
	                #li_StepCase := 240;
	            END_IF;

	        240: // Start sawing
	            "QX_MPO_M3_Saw_Q4" := TRUE;

	            #lx_Start_TON_Wait := TRUE;
	            #lt_TON_Wait := T#4000ms;

	            IF #lfb_TON_Wait.Q THEN
	                #li_Return_LDT := RD_SYS_T(#ldt_MQTT);
	                "gtyp_MPO".History[6].i_code := 600;
	                "gtyp_MPO".History[6].ldt_ts := DT_TO_LDT(#ldt_MQTT);

	                #lx_Start_TON_Wait := FALSE;
	                "QX_MPO_M3_Saw_Q4" := FALSE;
	                #li_StepCase := 250;
	            END_IF;

	        250: // Position turn table Pos Belt
	            IF "IX_MPO_RefSwitchTurnTable_PosSaw_I4" AND NOT "IX_MPO_RefSwitchTurnTable_PosBelt_I2" AND NOT "IX_MPO_RefSwitchTurnTable_PosVac_I1" THEN
	                "QX_MPO_M1_TurnTableClockwise_Q1" := TRUE;
	                "QX_MPO_M1_TurnTableCounterclockwise_Q2" := FALSE;
	            ELSIF NOT "IX_MPO_RefSwitchTurnTable_PosSaw_I4" AND "IX_MPO_RefSwitchTurnTable_PosBelt_I2" AND NOT "IX_MPO_RefSwitchTurnTable_PosVac_I1" THEN
	                "QX_MPO_M1_TurnTableClockwise_Q1" := FALSE;
	                "QX_MPO_M1_TurnTableCounterclockwise_Q2" := FALSE;
	                #li_StepCase := 260;
	            END_IF;

	        260: // put workpiece to belt
	            "QX_MPO_ValveFeeder_Q14" := TRUE;

	            #lx_Start_TON_Wait := TRUE;
	            #lt_TON_Wait := T#1000ms;

	            IF #lfb_TON_Wait.Q THEN
	                #lx_Start_TON_Wait := FALSE;
	                "QX_MPO_ValveFeeder_Q14" := FALSE;
	                "QX_MPO_Compressor_Q10" := FALSE;
	                #li_StepCase := 270;
	            END_IF;

	        270: // Position turn table Pos Vacuum
	            IF "IX_MPO_RefSwitchTurnTable_PosSaw_I4" OR "IX_MPO_RefSwitchTurnTable_PosBelt_I2" OR NOT "IX_MPO_RefSwitchTurnTable_PosVac_I1" THEN
	                "QX_MPO_M1_TurnTableClockwise_Q1" := FALSE;
	                "QX_MPO_M1_TurnTableCounterclockwise_Q2" := TRUE;
	            ELSIF NOT "IX_MPO_RefSwitchTurnTable_PosSaw_I4" AND NOT "IX_MPO_RefSwitchTurnTable_PosBelt_I2" AND "IX_MPO_RefSwitchTurnTable_PosVac_I1" THEN
	                "QX_MPO_M1_TurnTableClockwise_Q1" := FALSE;
	                "QX_MPO_M1_TurnTableCounterclockwise_Q2" := FALSE;
	                "QX_MPO_Compressor_Q10" := FALSE;
	                #li_StepCase := 280;
	            END_IF;

	        280: // Start conveyor belt
	            "QX_MPO_M2_ConveyorBeltForward_Q3" := TRUE;

	            #lx_Time_Error := TRUE;

	            IF #lfb_TOF_ConveyerBelt_Out.Q THEN
	                "gtyp_SLD".History  := "gtyp_MPO".History;
	                "gtyp_SLD".Workpiece := "gtyp_MPO".Workpiece;
	                "gtyp_MPO".Workpiece.s_id := '0';
	                "gtyp_MPO".Workpiece.s_state := '';
	                "gtyp_MPO".Workpiece.s_type := '';
	                FOR #li_Counter := 1 TO 8 DO
	                    "gtyp_MPO".History[#li_Counter].i_code := 0;
	                    "gtyp_MPO".History[#li_Counter].ldt_ts := DT#1990-01-01-00:00:00;
	                END_FOR;

	                "gtyp_Interface_Dashboard".Subscribe.State_MPO.x_active := FALSE;

	                #lx_Time_Error := FALSE;
	                #li_StepCase := 290;
	            END_IF;

	            // runtime error
	            IF #lfb_TON_Error.Q THEN
	                #li_Lights := 4;
	                #lx_Time_Error := FALSE;
	                "QX_MPO_M2_ConveyorBeltForward_Q3" := FALSE;
	                "gtyp_Interface_Dashboard".Subscribe.State_MPO.x_active := FALSE;
	                "gtyp_MPO".x_Error := TRUE;
	                #li_StepCase := 0;
	            END_IF;

	        290: // wait for runtime on conveyor belt

	            IF NOT #lfb_TOF_ConveyerBelt_Out.Q THEN
	                #lx_Start_TON_Wait := FALSE;
	                "QX_MPO_M2_ConveyorBeltForward_Q3" := FALSE;
	                #li_StepCase := 60;
	            END_IF;
	        // Statement section ELSE
	        ELSE
	            ;
	    END_CASE;

	    "QW_MPO_PWM_TurnTable_M1"   := "gtyp_MPO"."i_PWM_TurnTable";
	    "QW_MPO_PWM_Vacuum_M5"      := "gtyp_MPO"."i_PWM_Vacuum";

	ELSE
	    #li_Lights := 1;
	    #lx_Init := TRUE;
	    "gtyp_MPO".x_Start_Park_Position := FALSE;
	    "gtyp_MPO".x_Park_Position_Reached := FALSE;
	END_IF;
END_FUNCTION_BLOCK

FUNCTION_BLOCK "PRG_VGR_Axis_vertical"
TITLE = Program Axis vertical VGR
{ S7_Optimized_Access := 'TRUE' }
AUTHOR : 'A.Schaefer'
VERSION : 0.0
   VAR
      lx_Init { ExternalAccessible := 'False'; ExternalVisible := 'False'; ExternalWritable := 'False'} : Bool;
      lfb_vertical_Axis { ExternalAccessible := 'False'; ExternalVisible := 'False'; ExternalWritable := 'False'; S7_SetPoint := 'False'} : "FB_Axis";
   END_VAR


BEGIN
	IF #lx_Init THEN

	    // FB Axis vertical
	    #lfb_vertical_Axis(ini_Axis         := 2,
	                indi_Increment          := "gtyp_VGR".vertical_Axis.di_Increment,
	                inx_Ref_Switch          := "IX_VGR_RefSwitchVerticalAxis_I1",
	                inx_Referencing         := "gtyp_VGR".vertical_Axis.x_Reference,
	                inx_Start_Positioning   := "gtyp_VGR".vertical_Axis.x_Start_Positioning,
	                indi_Target_Position    := "gtyp_VGR".vertical_Axis.di_Target_Position,
	                ini_PWM                 := "gtyp_VGR".vertical_Axis.i_PWM,
	                inouttyp_Config         := "gtyp_VGR".vertical_Axis.Config,
	                inouttyp_Setup          := "gtyp_SetupAxis");

	    "QX_VGR_M1_VerticalAxisUp_Q1"       := #lfb_vertical_Axis.outx_Motor_Neg;
	    "QX_VGR_M1_VerticalAxisDown_Q2"     := #lfb_vertical_Axis.outx_Motor_Pos;
	    "QW_VGR_PWM_Vertical_M1"            := #lfb_vertical_Axis.outi_Motor_PWM;
	    "gtyp_VGR".vertical_Axis.di_Actual_Position:= #lfb_vertical_Axis.outdi_Actual_Position;
	    "gtyp_VGR".vertical_Axis.x_Referenced      := #lfb_vertical_Axis.outx_Referenced;
	    "gtyp_VGR".vertical_Axis.x_Position_Reached:= #lfb_vertical_Axis.outx_Position_Reached;
	ELSE
	    #lx_Init := TRUE;
	END_IF;
END_FUNCTION_BLOCK

FUNCTION_BLOCK "PRG_HBW_Axis_Vertical"
TITLE = Program Axis vertical HBW
{ S7_Optimized_Access := 'TRUE' }
AUTHOR : 'A.Schaefer'
VERSION : 0.0
   VAR
      lx_Init { ExternalAccessible := 'False'; ExternalVisible := 'False'; ExternalWritable := 'False'} : Bool;
      lfb_Vertical_Axis { ExternalAccessible := 'False'; ExternalVisible := 'False'; ExternalWritable := 'False'; S7_SetPoint := 'False'} : "FB_Axis";
   END_VAR


BEGIN
	IF #lx_Init THEN

	    // FB Axis vertical
	    #lfb_Vertical_Axis( ini_Axis                := 7,
	                        indi_Increment          := "gtyp_HBW".Vertical_Axis.di_Increment,
	                        inx_Ref_Switch          := "IX_HBW_RefSwitchVerticalAxis_I4",
	                        inx_Referencing         := "gtyp_HBW".Vertical_Axis.x_Reference,
	                        inx_Start_Positioning   := "gtyp_HBW".Vertical_Axis.x_Start_Positioning,
	                        indi_Target_Position    := "gtyp_HBW".Vertical_Axis.di_Target_Position,
	                        ini_PWM                 := "gtyp_HBW".Vertical_Axis.i_PWM,
	                        inouttyp_Config         := "gtyp_HBW".Vertical_Axis.Config,
	                        inouttyp_Setup          := "gtyp_SetupAxis");

	    "QX_HBW_M3_VerticalAxisDownward_Q5"           := #lfb_Vertical_Axis.outx_Motor_Pos;
	    "QX_HBW_M3_VerticalAxisUpward_Q6"             := #lfb_Vertical_Axis.outx_Motor_Neg;
	    "QW_HBW_PWM_VerticalAxis_M3"                  := #lfb_Vertical_Axis.outi_Motor_PWM;
	    "gtyp_HBW".Vertical_Axis.di_Actual_Position   := #lfb_Vertical_Axis.outdi_Actual_Position;
	    "gtyp_HBW".Vertical_Axis.x_Referenced         := #lfb_Vertical_Axis.outx_Referenced;
	    "gtyp_HBW".Vertical_Axis.x_Position_Reached   := #lfb_Vertical_Axis.outx_Position_Reached;
	ELSE
	    #lx_Init := TRUE;
	END_IF;
END_FUNCTION_BLOCK

